// ---- 20_Product/10_BCF/11_Conv/12_E_Functions/01_DUTs/ST_CFG_Zone.TcDUT
// Zone configuration structure
TYPE ST_CFG_Zone:
(**************************************************************************************
 * 	Application		:	BoxControl Framework
 *	Revision		:	$Revision: 474969 $
 *	Revision date	:	$Date: 2021-04-08 19:53:18 +0200 (tor, 08 apr 2021) $
 *	Last changed by	:	$Author: d7mangc $
 *	URL				:	$URL: http://almscdc.swisslog.com/repo/SWPD/Development/BoxControlFramework/20_Release/tags/R1.12.0/01_Software/BCF/BCF/JumpStart/20_Product/10_BCF/11_Conv/12_E_Functions/01_DUTs/ST_CFG_Zone.TcDUT $
 *
 *	Purpose			:	Zone configuration - contains the configuration for a zone.
 *
 * ------------------------------------------------------------------------------------
 *	Copyright Swisslog [IP AG], Switzerland. All rights reserved.
 * 
 * ------------------------------------------------------------------------------------
 *	
 * 	Revision History: 
 *
 * VERSION DATE         INITIALS     DESCRIPTION
 * 0.0     DD.MM.YYYY   (name)       (explain customized modifications)
 *
 **************************************************************************************)
STRUCT
	ZoneName						: STRING[NAME_LENGTH]	:= 'MM-GGG-EEEE-FF-Z';			// Name of the zone
	Length							: ARRAY[1..3] OF UINT	:= [1000, 0, 0];				// Length of the zone based on the transport direction [mm]
	//-----------------------------------------------------------------------------------------------
	Speed							: REAL					:= 1.0;							// Maximal speed of the zone [m/s]
	SpeedSlow						: INT					:=  50;							// Speed slow [%]
	SpeedFast						: INT					:= 100;							// Speed fast [%]
	SpeedRatio						: REAL					:= 1/1;							// Transmission ratio between speed command and movement speed of the TU
	//-----------------------------------------------------------------------------------------------
	EnablePrestart					: BOOL					:= TRUE;						// Enable prestart drive two zones ahead
	EnableFreeRun					: BOOL					:= TRUE;						// Enable free run
	EnableMultipleTU_Transition		: BOOL					:= FALSE;						// Enable multiple TU transition
	EnableJamAutoReset				: BOOL					:= TRUE;						// Enable jam auto reset if signal is free
	EnableMFC						: BOOL					:= FALSE;						// Enable material flow control
	EnableIgnoreNextZoneState		: BOOL					:= FALSE;						// Enable ignore the state of the next zone at handover
	EnableSimultaneousTransport		: BOOL					:= FALSE;						// Enable simultaneous transport
	EnableLowPressureAccumulation	: BOOL					:= FALSE;						// Enable low pressure accumulation - NOT IMPLEMENTED -
	EnableSlugRelease				: BOOL					:= FALSE;						// Enable slug release -NOT IMPLEMENTED -
	EnableFastSpeed					: BOOL					:= TRUE;						// Enable fast speed 
	EnableMultizone					: BOOL					:= TRUE;						// Enable multizone
	EnableCreateGapOnlyAtRestart	: BOOL					:= FALSE;						// Enable create gap only when drive restarts
	EnableLatchOccupiedState		: BOOL					:= FALSE;						// Enable latch occupied state
	EnableRoutingUpdate             : BOOL                  := FALSE;						// Enable routing update
	EnableAddOnSensor               : BOOL    				:= FALSE;						// Will use the sensor from the addon interface
    EnableMotorControl              : BOOL                  := FALSE;                       // Needs to be enabled for the zones using common motor with slugging
	//-----------------------------------------------------------------------------------------------
	SendTransportTaskCompleted		: BOOL					:= FALSE;						// Send a transport complete report if destination is reached
	SendTransportTaskCompletedOcc	: BOOL					:= FALSE;						// Send a transport complete report if destination is reached and zone occupied
	SendPositionClear				: BOOL					:= FALSE;						// Send a position clear report if zone is physically free
	SendPositionOccupied			: BOOL					:= FALSE;						// Send a position pccupied report if zone is physically occupied
	SendIdentificationReport		: BOOL					:= FALSE;						// Send an identification point report if zone is physically occupied
	eTUR_SendMode					: E_TUR_SendModes		:= E_TUR_SendModes.ALWAYS;		// Additional controls over when TUR is sent on TU index deletion for the zone 
	//-----------------------------------------------------------------------------------------------
	AddTU_Data						: BOOL					:= FALSE;						// Add TU data 
	DeleteTU_DataTakeOver			: BOOL					:= FALSE;						// Delete TU data at takeover
	DeleteTU_DataZoneFree			: BOOL					:= FALSE;						// Delete TU data if the zone is free
	//-----------------------------------------------------------------------------------------------
	tZoneFree						: TIME					:= T#0S;						// Delay time for zone free, if 0 then standard value will be used (2s)
	tZoneOccupied					: TIME					:= T#0S;						// Delay time for zone occupied, if 0 then standard value will be used (2s)
	ClearingDistance				: UINT					:= 2_000;						// Clearing distance [mm]
	JamTriggerDistance				: UINT					:= 2_000;						// Driving distance after jam error is triggered [mm]
	TimeoutTakeDistance				: UINT					:= 0;							// Driving distance after timeout take is triggered, if 0 then calculated value will be used [mm]
	MinimumTU_Distance				: UINT					:= 0;							// Delays the takeover to ensure this minimum gap between the TU’s [mm]
	TakeoverPlausibilityDistance	: UINT					:= 0;							// Distance for takeover plausibility check, if 0 then calculated value will be used [mm] 
	StopDelayDistanceFromSide		: ARRAY[1..4] OF UINT	:= [  0,   0,   0,   0];		// Stop distance after occupied signal [mm]
    tTakeoverMotorStartDelay        : TIME                  := T#0S;						// Delay before starting the motor on takeover (slugging)
	ZoneEndLengthToSide				: ARRAY[1..4] OF UINT	:= [100, 100, 100, 100];		// Length between occupied signal and zone end [mm]
END_STRUCT
END_TYPE

// ---- 20_Product/10_BCF/11_Conv/12_E_Functions/01_DUTs/ST_CM_ZoneBase.TcDUT
TYPE ST_CM_ZoneBase :
(**************************************************************************************
 * 	Application		:	BoxControl Framework
 *	Revision		:	$Revision: 404529 $
 *	Revision date	:	$Date: 2018-04-23 08:21:38 +0200 (Mo., 23 Apr 2018) $
 *	Last changed by	:	$Author: b7bolm $
 *	URL				:	$URL: http://almscdc.swisslog.com/repo/SWPD/Development/BoxControlFramework/20_Release/trunk/01_Software/BCF/BCF/JumpStart/20_Product/10_App/12_E_Functions/10_Lib/10_Conv/01_DUTs/ST_CM_ZoneBase.TcDUT $
 *
 *	Purpose			:	Base Structure for Condition monitoring 					
 *
 *
 * ------------------------------------------------------------------------------------
 *	Copyright Swisslog [IP AG], Switzerland. All rights reserved.
 * 
 * ------------------------------------------------------------------------------------
 *	
 * 	Revision History: 
 *
 * 	VERSION			DATE			INITIALS			DESCRIPTION
 *	0.1				01.01.2001		swl					Example
 *
 **************************************************************************************)	
STRUCT
	nCurrentTime 	: ULINT; // Current DC-Time of the PLC-Task
	Data			: ARRAY[E_CM_Index.E_BEGIN_VARIABLE+1..E_CM_Index.E_END_VARIABLE-1] OF ST_CM_GeneralData; //Process Data used by Condiition Monitoring Method 
	Settings		: ARRAY[E_CM_Index.E_BEGIN_VARIABLE+1..E_CM_Index.E_END_VARIABLE-1] OF ST_CM_Settings; //Settings Data set by Telegram/User
	
END_STRUCT
END_TYPE

// ---- 20_Product/10_BCF/11_Conv/12_E_Functions/01_DUTs/ST_FunctionBase.TcDUT
TYPE ST_FunctionBase :
(**************************************************************************************
 * 	Application		:	BoxControl Framework
 *	Revision		:	$Revision: 404529 $
 *	Revision date	:	$Date: 2018-04-23 08:21:38 +0200 (Mo., 23 Apr 2018) $
 *	Last changed by	:	$Author: b7bolm $
 *	URL				:	$URL: http://almscdc.swisslog.com/repo/SWPD/Development/BoxControlFramework/20_Release/trunk/01_Software/BCF/BCF/JumpStart/20_Product/10_App/12_E_Functions/10_Lib/10_Conv/01_DUTs/ST_FunctionBase.TcDUT $
 *
 *	Purpose			:	Function interface - Contains data which is provided by the
 *						function or is input from other objects.
 *
 * ------------------------------------------------------------------------------------
 *	Copyright Swisslog [IP AG], Switzerland. All rights reserved.
 * 
 * ------------------------------------------------------------------------------------
 *	
 * 	Revision History: 
 *
 * 	VERSION			DATE			INITIALS			DESCRIPTION
 *	0.1				01.01.2001		swl					Example
 *
 **************************************************************************************)
STRUCT
	AddOnAck					: BOOL; // Addon acknowledge
	STI_Instance				: ITF_SubsystemTransport; // Instance to compare valid interfaces
	eMsgType					: E_ITC_MsgTypeConv;
	Position					: ST_PositionIdent; // Position idents
	NextPositionName			: STRING(NAME_LENGTH); // Position idents
	PrevPositionName			: STRING(NAME_LENGTH); // Position idents
	PositionName				: STRING(NAME_LENGTH); // Position name
	DestinationName				: STRING(NAME_LENGTH); // Position name
	TU_DataIndex				: DINT; // Data index
	ErrorDataSet				: ST_ErrorDataSet; // Temporary error set
	ErrorDataZone				: ST_ZoneErrorStruct; // Temporary error data
	eReturnCode					: E_ErrorConv;
	DataITC						: ST_ITC_GeneralData; // ITC Message
	OperatingState				: ST_PositionState; // States
	LinkedFunctionStopped		: BOOL; // Linked function stopped
	AllZonesStopped				: BOOL; // All zones are stopped
	TransportControlParam		: ST_TransportControlParam; // Transportcontrol param
	TransportData				: ST_TransportData; // Transport data
	PrevTransportData			: ST_TransportData; // Previous data
	NextTransportData			: ST_TransportData; // Next data
	TransportDataEmpty			: ST_TransportData; // Transport data
	TransportControlDataEmpty 	: ST_TransportControlData; // Transport control data
	ZoneSettingsEmpty			: ST_CFG_Zone; // Zone settings
	PositionStateEmpty			: ST_PositionState;
	Idx							: INT; // iterator
	FSQ							: ST_ITC_FSQ; // ITC Message
	FCQ							: ST_ITC_FCQ; // ITC Message
	MCQ							: ST_ITC_MCQ; // ITC Message
	SIQ							: ST_ITC_SIQ; // ITC Message
	DAQ							: ST_ITC_DAQ; // ITC Message
	GDQ							: ST_ITC_GDQ; // ITC Message
	RAA							: ST_ITC_RAA; // ITC Message
	RDQ							: ST_ITC_RDQ; // ITC Message
	CM_Zone						: ARRAY [1..NUMBER_OF_ZONES_PER_FUNCTION] OF ST_CM_Base;	/// Data Aquisition Variables Staorage and Settings // CM inside base
END_STRUCT
END_TYPE

// ---- 20_Product/10_BCF/11_Conv/12_E_Functions/01_DUTs/ST_FunctionData.TcDUT
TYPE ST_FunctionData :
(**************************************************************************************
 * 	Application		:	BoxControl Framework
 *	Revision		:	$Revision: 404529 $
 *	Revision date	:	$Date: 2018-04-23 08:21:38 +0200 (Mo., 23 Apr 2018) $
 *	Last changed by	:	$Author: b7bolm $
 *	URL				:	$URL: http://almscdc.swisslog.com/repo/SWPD/Development/BoxControlFramework/20_Release/trunk/01_Software/BCF/BCF/JumpStart/20_Product/10_App/12_E_Functions/10_Lib/10_Conv/01_DUTs/ST_FunctionData.TcDUT $
 *
 *	Purpose			:	Function data
 *
 * ------------------------------------------------------------------------------------
 *	Copyright Swisslog [IP AG], Switzerland. All rights reserved.
 * 
 * ------------------------------------------------------------------------------------
 *	
 * 	Revision History: 
 *
 * 	VERSION			DATE			INITIALS			DESCRIPTION
 *	0.1				01.01.2001		swl					Example
 *
 **************************************************************************************)
STRUCT
	Init				: BOOL; // Initialized
	InitRunning			: BOOL; // Init ongoing
	OperationState		: ST_PositionState; // Information about the state
	AddOn				: ST_AddOnResult; // Result form external addons
	MemberList			: ST_FunctionMemberList; // List of members belonging to this function
	ErrorData			: ST_FunctionErrorStruct; // Error structure
	AddOnData			: ST_AddOnData; // Specific addon data structs
	ControlRequest		: ST_ControlRequest; // Control request
END_STRUCT
END_TYPE

// ---- 20_Product/10_BCF/11_Conv/12_E_Functions/01_DUTs/ST_FunctionElement.TcDUT
TYPE ST_FunctionElement :
(**************************************************************************************
 * 	Application		:	BoxControl Framework
 *	Revision		:	$Revision: 404529 $
 *	Revision date	:	$Date: 2018-04-23 08:21:38 +0200 (Mo., 23 Apr 2018) $
 *	Last changed by	:	$Author: b7bolm $
 *	URL				:	$URL: http://almscdc.swisslog.com/repo/SWPD/Development/BoxControlFramework/20_Release/trunk/01_Software/BCF/BCF/JumpStart/20_Product/10_App/12_E_Functions/10_Lib/10_Conv/01_DUTs/ST_FunctionElement.TcDUT $
 *
 *	Purpose			:	Function element
 *
 * ------------------------------------------------------------------------------------
 *	Copyright Swisslog [IP AG], Switzerland. All rights reserved.
 * 
 * ------------------------------------------------------------------------------------
 *	
 * 	Revision History: 
 *
 * 	VERSION			DATE			INITIALS			DESCRIPTION
 *	0.1				01.01.2001		swl					Example
 *
 **************************************************************************************)	
STRUCT
	OperationState	: ST_PositionState;
	State			: ST_ElementState;
END_STRUCT
END_TYPE

// ---- 20_Product/10_BCF/11_Conv/12_E_Functions/01_DUTs/ST_FunctionErrorStruct.TcDUT
TYPE ST_FunctionErrorStruct :
(**************************************************************************************
 * 	Application		:	BoxControl Framework
 *	Revision		:	$Revision: 404529 $
 *	Revision date	:	$Date: 2018-04-23 08:21:38 +0200 (Mo., 23 Apr 2018) $
 *	Last changed by	:	$Author: b7bolm $
 *	URL				:	$URL: http://almscdc.swisslog.com/repo/SWPD/Development/BoxControlFramework/20_Release/trunk/01_Software/BCF/BCF/JumpStart/20_Product/10_App/12_E_Functions/10_Lib/10_Conv/01_DUTs/ST_FunctionErrorStruct.TcDUT $
 *
 *	Purpose			:	Function error structure - Contains all information for the
 *						error handling.
 *
 * ------------------------------------------------------------------------------------
 *	Copyright Swisslog [IP AG], Switzerland. All rights reserved.
 * 
 * ------------------------------------------------------------------------------------
 *	
 * 	Revision History: 
 *
 * 	VERSION			DATE			INITIALS			DESCRIPTION
 *	0.1				01.01.2001		swl					Example
 *
 **************************************************************************************)
STRUCT
	ErrorState				: E_ErrorState; // Ongoing module error state
	Error					: ST_ErrorDataSet; // Ongoing reported function error
	DataSetIdx				: INT; // Choosen error set index
	ErrorDataSet			: ARRAY [1..NUMBER_OF_ERROR_SETS] OF ST_ErrorDataSet; // Overview about all message sets
	ExternalError			: ST_ErrorDataSet; // External error, Can be set customized or by control code
	ZoneErrorPending		: BOOL; // A zone of this function is in error state
END_STRUCT
END_TYPE

// ---- 20_Product/10_BCF/11_Conv/12_E_Functions/01_DUTs/ST_FunctionInterface.TcDUT
TYPE ST_FunctionInterface :
(**************************************************************************************
 * 	Application		:	BoxControl Framework
 *	Revision		:	$Revision: 404529 $
 *	Revision date	:	$Date: 2018-04-23 08:21:38 +0200 (Mo., 23 Apr 2018) $
 *	Last changed by	:	$Author: b7bolm $
 *	URL				:	$URL: http://almscdc.swisslog.com/repo/SWPD/Development/BoxControlFramework/20_Release/trunk/01_Software/BCF/BCF/JumpStart/20_Product/10_App/12_E_Functions/10_Lib/10_Conv/01_DUTs/ST_FunctionInterface.TcDUT $
 *
 *	Purpose			:	Function interface - Contains data which is provided by the
 *						function or is input from other objects.
 *
 * ------------------------------------------------------------------------------------
 *	Copyright Swisslog [IP AG], Switzerland. All rights reserved.
 * 
 * ------------------------------------------------------------------------------------
 *	
 * 	Revision History: 
 *
 * 	VERSION			DATE			INITIALS			DESCRIPTION
 *	0.1				01.01.2001		swl					Example
 *
 **************************************************************************************)
STRUCT
	In		: ST_FunctionInterfaceIn;
	Out		: ST_FunctionInterfaceOut;
END_STRUCT
END_TYPE

// ---- 20_Product/10_BCF/11_Conv/12_E_Functions/01_DUTs/ST_FunctionInterfaceIn.TcDUT
TYPE ST_FunctionInterfaceIn :
(**************************************************************************************
 * 	Application		:	BoxControl Framework
 *	Revision		:	$Revision: 404529 $
 *	Revision date	:	$Date: 2018-04-23 08:21:38 +0200 (Mo., 23 Apr 2018) $
 *	Last changed by	:	$Author: b7bolm $
 *	URL				:	$URL: http://almscdc.swisslog.com/repo/SWPD/Development/BoxControlFramework/20_Release/trunk/01_Software/BCF/BCF/JumpStart/20_Product/10_App/12_E_Functions/10_Lib/10_Conv/01_DUTs/ST_FunctionInterfaceIn.TcDUT $
 *
 *	Purpose			:	Function interface - Contains data which is provided by the
 *						function or is input from other objects.
 *
 * ------------------------------------------------------------------------------------
 *	Copyright Swisslog [IP AG], Switzerland. All rights reserved.
 * 
 * ------------------------------------------------------------------------------------
 *	
 * 	Revision History: 
 *
 * 	VERSION			DATE			INITIALS			DESCRIPTION
 *	0.1				01.01.2001		swl					Example
 *
 **************************************************************************************)
STRUCT
	ePrevFunctionNumber 	: E_FunctionNumber; // Previous element function number
	eNextFunctionNumber 	: E_FunctionNumber; // Next element function number	
	FunctionEnable			: BOOL := TRUE; // External function enable 
	Element					: ST_FunctionElement; // States of the function corresponding element
	AddOnOrder				: ARRAY [1..Conveyor.NUMBER_OF_ADDON_FUNCTIONS] OF ST_AddOn; // Number of addons per function
END_STRUCT
END_TYPE

// ---- 20_Product/10_BCF/11_Conv/12_E_Functions/01_DUTs/ST_FunctionInterfaceOut.TcDUT
TYPE ST_FunctionInterfaceOut :
(**************************************************************************************
 * 	Application		:	BoxControl Framework
 *	Revision		:	$Revision: 404529 $
 *	Revision date	:	$Date: 2018-04-23 08:21:38 +0200 (Mo., 23 Apr 2018) $
 *	Last changed by	:	$Author: b7bolm $
 *	URL				:	$URL: http://almscdc.swisslog.com/repo/SWPD/Development/BoxControlFramework/20_Release/trunk/01_Software/BCF/BCF/JumpStart/20_Product/10_App/12_E_Functions/10_Lib/10_Conv/01_DUTs/ST_FunctionInterfaceOut.TcDUT $
 *
 *	Purpose			:	Function interface - Contains data which is provided by the
 *						function or is input from other objects.
 *
 * ------------------------------------------------------------------------------------
 *	Copyright Swisslog [IP AG], Switzerland. All rights reserved.
 * 
 * ------------------------------------------------------------------------------------
 *	
 * 	Revision History: 
 *
 * 	VERSION			DATE			INITIALS			DESCRIPTION
 *	0.1				01.01.2001		swl					Example
 *
 **************************************************************************************)
STRUCT
	FunctionOrders		: ST_FunctionOrders; // Function orders to the element
	AddOnOrders			: ST_AddOnOrders; // AddOn orders
	Interlock			: ST_Interlock; // Interlock structure
END_STRUCT
END_TYPE

// ---- 20_Product/10_BCF/11_Conv/12_E_Functions/01_DUTs/ST_FunctionMemberList.TcDUT
TYPE ST_FunctionMemberList :
(**************************************************************************************
 * 	Application		:	BoxControl Framework
 *	Revision		:	$Revision: 404529 $
 *	Revision date	:	$Date: 2018-04-23 08:21:38 +0200 (Mo., 23 Apr 2018) $
 *	Last changed by	:	$Author: b7bolm $
 *	URL				:	$URL: http://almscdc.swisslog.com/repo/SWPD/Development/BoxControlFramework/20_Release/trunk/01_Software/BCF/BCF/JumpStart/20_Product/10_App/12_E_Functions/10_Lib/10_Conv/01_DUTs/ST_FunctionMemberList.TcDUT $
 *
 *	Purpose			:	Function member list - Contains all objects belonging to this 
 *						function.
 *
 * ------------------------------------------------------------------------------------
 *	Copyright Swisslog [IP AG], Switzerland. All rights reserved.
 * 
 * ------------------------------------------------------------------------------------
 *	
 * 	Revision History: 
 *
 * 	VERSION			DATE			INITIALS			DESCRIPTION
 *	0.1				01.01.2001		swl					Example
 *
 **************************************************************************************)
STRUCT
	AddOnList		: ARRAY [1 .. NUMBER_OF_ADDON_FUNCTIONS] OF ST_AddonEntry;
END_STRUCT
END_TYPE

// ---- 20_Product/10_BCF/11_Conv/12_E_Functions/01_DUTs/ST_FunctionOrders.TcDUT
///Element function order - This structure serves as order command to the function related element.
TYPE ST_FunctionOrders :
(**************************************************************************************
 *  Application     :   BoxControl Framework
 *  Revision date   :   $Date: 2013-09-23 11:26:06 +0200 (Wed, 23 Sep 2015) $
 *  Author          :   CDC
 * ------------------------------------------------------------------------------------
 *  © Swisslog AG
 *  Swisslog is not liable for any usage of this source code that is not agreed 
 *  on between Swisslog and the other party. The mandatory legal liability remains 
 *  unaffected.
 * ------------------------------------------------------------------------------------
 *  Revision History: 
 *
 *  VERSION DATE         INITIALS     DESCRIPTION
 *  0.0     DD.MM.YYYY   (name)       (explain customized modifications)
 *
 **************************************************************************************)
 //Comment changed according to BCFD-6292 - ST_FunctionOrders, Comments not correct	
STRUCT
    //Axis 1 <-> 2
	Enable				: BOOL; // Function enables transport
	ReqDriveRun			: BOOL; // Request for drive run
	ReqDriveDirection	    : BOOL; // Request drive direction. TRUE = 1->2, False 2->1
	ReqSpeed			: INT; // Request for this speed

    //Axis 3 <-> 4
	Enable_34				: BOOL; // Function enables transport
	ReqDriveRun_34			: BOOL; // Request for drive run
	ReqSpeed_34				: INT; // Request for speed	
	ReqDriveDirection_34	: BOOL; // Request drive direction. True = 3->4, False = 4->3
END_STRUCT
END_TYPE

// ---- 20_Product/10_BCF/11_Conv/12_E_Functions/01_DUTs/ST_ITC_Function.TcDUT
TYPE ST_ITC_Function :
(**************************************************************************************
 * 	Application		:	BoxControl Framework
 *	Revision		:	$Revision: 404529 $
 *	Revision date	:	$Date: 2018-04-23 08:21:38 +0200 (Mo., 23 Apr 2018) $
 *	Last changed by	:	$Author: b7bolm $
 *	URL				:	$URL: http://almscdc.swisslog.com/repo/SWPD/Development/BoxControlFramework/20_Release/trunk/01_Software/BCF/BCF/JumpStart/20_Product/10_App/12_E_Functions/10_Lib/10_Conv/01_DUTs/ST_ITC_Function.TcDUT $
 *
 *	Purpose			:	Function ITC structure
 *
 * ------------------------------------------------------------------------------------
 *	Copyright Swisslog [IP AG], Switzerland. All rights reserved.
 * 
 * ------------------------------------------------------------------------------------
 *	
 * 	Revision History: 
 *
 * 	VERSION			DATE			INITIALS			DESCRIPTION
 *	0.1				01.01.2001		swl					Example
 *
 **************************************************************************************)
STRUCT
	FunctionITC		: ST_ITC_FunctionITC; // ITC function data
	ZoneITC			: ARRAY [1..NUMBER_OF_ZONES_PER_FUNCTION] OF ST_ITC_Zone; // ITC Zone data
	ManualMotion	: ST_ITC_ManualMotion; // Command for manual motion
END_STRUCT
END_TYPE

// ---- 20_Product/10_BCF/11_Conv/12_E_Functions/01_DUTs/ST_ITC_FunctionCommands.TcDUT
TYPE ST_ITC_FunctionCommands :
(**************************************************************************************
 * 	Application		:	BoxControl Framework
 *	Revision		:	$Revision: 404529 $
 *	Revision date	:	$Date: 2018-04-23 08:21:38 +0200 (Mo., 23 Apr 2018) $
 *	Last changed by	:	$Author: b7bolm $
 *	URL				:	$URL: http://almscdc.swisslog.com/repo/SWPD/Development/BoxControlFramework/20_Release/trunk/01_Software/BCF/BCF/JumpStart/20_Product/10_App/12_E_Functions/10_Lib/10_Conv/01_DUTs/ST_ITC_FunctionCommands.TcDUT $
 *
 *	Purpose			:	Internal ITC function commands
 *
 * ------------------------------------------------------------------------------------
 *	Copyright Swisslog [IP AG], Switzerland. All rights reserved.
 * 
 * ------------------------------------------------------------------------------------
 *	
 * 	Revision History: 
 *
 * 	VERSION			DATE			INITIALS			DESCRIPTION
 *	0.1				01.01.2001		swl					Example
 *
 **************************************************************************************)
STRUCT
	StatusReport			: BOOL; // Command to send StatusReport 
	ControlReport			: BOOL; // Command to send ControlReport 
	NoErrorReport			: BOOL; // Command to send a 'no error' report
	ManualControlReport		: BOOL; // Command to send a manual control report
	ScannerInformationReport: BOOL; // Command to send a scanner information report
	ScannerNoReadReport		: BOOL; // Command to send a scanner no read report
END_STRUCT
END_TYPE

// ---- 20_Product/10_BCF/11_Conv/12_E_Functions/01_DUTs/ST_ITC_FunctionITC.TcDUT
TYPE ST_ITC_FunctionITC :
(**************************************************************************************
 * 	Application		:	BoxControl Framework
 *	Revision		:	$Revision: 404529 $
 *	Revision date	:	$Date: 2018-04-23 08:21:38 +0200 (Mo., 23 Apr 2018) $
 *	Last changed by	:	$Author: b7bolm $
 *	URL				:	$URL: http://almscdc.swisslog.com/repo/SWPD/Development/BoxControlFramework/20_Release/trunk/01_Software/BCF/BCF/JumpStart/20_Product/10_App/12_E_Functions/10_Lib/10_Conv/01_DUTs/ST_ITC_FunctionITC.TcDUT $
 *
 *	Purpose			:	Function ITC structure
 *
 * ------------------------------------------------------------------------------------
 *	Copyright Swisslog [IP AG], Switzerland. All rights reserved.
 * 
 * ------------------------------------------------------------------------------------
 *	
 * 	Revision History: 
 *
 * 	VERSION			DATE			INITIALS			DESCRIPTION
 *	0.1				01.01.2001		swl					Example
 *
 **************************************************************************************)
STRUCT
	Commands		: ST_ITC_FunctionCommands; // Internal ITC commands
	Variable		: DINT; // Control variable
END_STRUCT
END_TYPE

// ---- 20_Product/10_BCF/11_Conv/12_E_Functions/01_DUTs/ST_ITC_Zone.TcDUT
TYPE ST_ITC_Zone :
(**************************************************************************************
 * 	Application		:	BoxControl Framework
 *	Revision		:	$Revision: 404529 $
 *	Revision date	:	$Date: 2018-04-23 08:21:38 +0200 (Mo., 23 Apr 2018) $
 *	Last changed by	:	$Author: b7bolm $
 *	URL				:	$URL: http://almscdc.swisslog.com/repo/SWPD/Development/BoxControlFramework/20_Release/trunk/01_Software/BCF/BCF/JumpStart/20_Product/10_App/12_E_Functions/10_Lib/10_Conv/01_DUTs/ST_ITC_Zone.TcDUT $
 *
 *	Purpose			:	Zone ITC structures
 *
 * ------------------------------------------------------------------------------------
 *	Copyright Swisslog [IP AG], Switzerland. All rights reserved.
 * 
 * ------------------------------------------------------------------------------------
 *	
 * 	Revision History: 
 *
 * 	VERSION			DATE			INITIALS			DESCRIPTION
 *	0.1				01.01.2001		swl					Example
 *
 **************************************************************************************)
STRUCT
	Commands	: ST_ITC_ZoneCommands; // Internal zone ITC commands
	Variable	: DINT; // Control variable
	Flags		: ST_ITC_ZoneFlags; // Flags
END_STRUCT
END_TYPE

// ---- 20_Product/10_BCF/11_Conv/12_E_Functions/01_DUTs/ST_ITC_ZoneCommands.TcDUT
TYPE ST_ITC_ZoneCommands :
(**************************************************************************************
 * 	Application		:	BoxControl Framework
 *	Revision		:	$Revision: 404529 $
 *	Revision date	:	$Date: 2018-04-23 08:21:38 +0200 (Mo., 23 Apr 2018) $
 *	Last changed by	:	$Author: b7bolm $
 *	URL				:	$URL: http://almscdc.swisslog.com/repo/SWPD/Development/BoxControlFramework/20_Release/trunk/01_Software/BCF/BCF/JumpStart/20_Product/10_App/12_E_Functions/10_Lib/10_Conv/01_DUTs/ST_ITC_ZoneCommands.TcDUT $
 *
 *	Purpose			:	Zone commands
 *
 * ------------------------------------------------------------------------------------
 *	Copyright Swisslog [IP AG], Switzerland. All rights reserved.
 * 
 * ------------------------------------------------------------------------------------
 *	
 * 	Revision History: 
 *
 * 	VERSION			DATE			INITIALS			DESCRIPTION
 *	0.1				01.01.2001		swl					Example
 *
 **************************************************************************************)	
STRUCT
	NoErrorReport				: BOOL; // Command to send a no error report 
	StatusReport				: BOOL; // Command to send a status report 
	ControlReport				: BOOL; // Command TO send a control report 
	TransportTaskCompleted		: BOOL; // Command to send a transport task report 
	PositionOccupied			: BOOL; // Command to send a position occupied report 
	PositionCleared				: BOOL; // Command to send a position cleared report 
	IdentificationReport		: BOOL; // Command to send an identification point report
END_STRUCT
END_TYPE

// ---- 20_Product/10_BCF/11_Conv/12_E_Functions/01_DUTs/ST_ITC_ZoneFlags.TcDUT
TYPE ST_ITC_ZoneFlags :
(**************************************************************************************
 * 	Application		:	BoxControl Framework
 *	Revision		:	$Revision: 404529 $
 *	Revision date	:	$Date: 2018-04-23 08:21:38 +0200 (Mo., 23 Apr 2018) $
 *	Last changed by	:	$Author: b7bolm $
 *	URL				:	$URL: http://almscdc.swisslog.com/repo/SWPD/Development/BoxControlFramework/20_Release/trunk/01_Software/BCF/BCF/JumpStart/20_Product/10_App/12_E_Functions/10_Lib/10_Conv/01_DUTs/ST_ITC_ZoneFlags.TcDUT $
 *
 *	Purpose			:	Zone flags
 *
 * ------------------------------------------------------------------------------------
 *	Copyright Swisslog [IP AG], Switzerland. All rights reserved.
 * 
 * ------------------------------------------------------------------------------------
 *	
 * 	Revision History: 
 *
 * 	VERSION			DATE			INITIALS			DESCRIPTION
 *	0.1				01.01.2001		swl					Example
 *
 **************************************************************************************)	
STRUCT
	TransportTaksCompleteOccSent	: BOOL; // Store sent information
	TransportTaksCompleteSent		: BOOL; // Store sent information
	PositionClearSent				: BOOL; // Store sent information
	PositionOccupiedSent			: BOOL; // Store sent information
	IdentificationReportSent		: BOOL; // Store sent information
END_STRUCT
END_TYPE

// ---- 20_Product/10_BCF/11_Conv/12_E_Functions/01_DUTs/ST_LastTUdata.TcDUT
TYPE ST_LastTUdata :
STRUCT
	TU_ID			: STRING(Conveyor.TU_ID_STRINGLENGTH); // TU_ID as characters 1 to 18 
  	AssignmentID	: UDINT; // Assignment ID
  	TU_Type			: INT; // Type of transport unit 
END_STRUCT
END_TYPE

// ---- 20_Product/10_BCF/11_Conv/12_E_Functions/01_DUTs/ST_TransportControlData.TcDUT
TYPE ST_TransportControlData :
(**************************************************************************************
 * 	Application		:	BoxControl Framework
 *	Revision		:	$Revision: 404529 $
 *	Revision date	:	$Date: 2018-04-23 08:21:38 +0200 (Mo., 23 Apr 2018) $
 *	Last changed by	:	$Author: b7bolm $
 *	URL				:	$URL: http://almscdc.swisslog.com/repo/SWPD/Development/BoxControlFramework/20_Release/trunk/01_Software/BCF/BCF/JumpStart/20_Product/10_App/12_E_Functions/10_Lib/10_Conv/01_DUTs/ST_TransportControlData.TcDUT $
 *
 *	Purpose			:	Transport control
 *
 * ------------------------------------------------------------------------------------
 *	Copyright Swisslog [IP AG], Switzerland. All rights reserved.
 * 
 * ------------------------------------------------------------------------------------
 *	
 * 	Revision History: 
 *
 * 	VERSION			DATE			INITIALS			DESCRIPTION
 *	0.1				01.01.2001		swl					Example
 *
 **************************************************************************************)	
STRUCT
	eTransportState					: E_TransportState		:= E_TransportState.UNDEFINED;	// Transport state
	eTakeOverState 					: E_TakeOverState		:= E_TakeOverState.UNDEFINED;	// Takeover state
	eHandOverState 					: E_HandOverState		:= E_HandOverState.UNDEFINED;	// Handover state
	TransportParam					: ST_TransportParam;									// Transport parameter valid for current transport
	//-----------------------------------------------------------------------------------------------
	Occupied						: BOOL					:= FALSE; 						// Position is physically occupied
	DataPresent						: BOOL					:= FALSE;						// Position is logically occupied
	TU_DataIndex					: DINT					:= 0;							// Current TU data index
	LastTU_DataIndex 				: DINT					:= 0;							// Last TU data index
	NumberOfPresentTUs  			: UINT					:= 0;							// Number of present TUs on this zone (the TU in handover is counted by the next zone)
	FastSpeedActive					: BOOL					:= FALSE;						// Fast speed is active
	DriveRunning					: BOOL					:= FALSE;						// Drive is running
	MovementPosition				: UDINT					:= 0;							// Movement position value [mm]	
	Stopped							: BOOL					:= FALSE;						// Module is stopped
	SensorOccupied      			: BOOL					:= FALSE;						// Sensor position occupied
	TransportActive     			: BOOL					:= FALSE;						// Transport is active
	//-----------------------------------------------------------------------------------------------
	CurrentSpeed					: INT					:= 0;							// Current speed
	LimitSpeedToPrev				: INT					:= 0;							// Current valid speed limit to previous zone
	LimitSpeedToNext				: INT					:= 0;							// Current valid speed limit to next zone
	//-----------------------------------------------------------------------------------------------
	TU_LeadingEdgePos				: DINT					:= 0;							// TU leading edge position [mm]
END_STRUCT
END_TYPE

// ---- 20_Product/10_BCF/11_Conv/12_E_Functions/01_DUTs/ST_TransportControlParam.TcDUT
TYPE ST_TransportControlParam :
(**************************************************************************************
 * 	Application		:	BoxControl Framework
 *	Revision		:	$Revision: 404529 $
 *	Revision date	:	$Date: 2018-04-23 08:21:38 +0200 (Mo., 23 Apr 2018) $
 *	Last changed by	:	$Author: b7bolm $
 *	URL				:	$URL: http://almscdc.swisslog.com/repo/SWPD/Development/BoxControlFramework/20_Release/trunk/01_Software/BCF/BCF/JumpStart/20_Product/10_App/12_E_Functions/10_Lib/10_Conv/01_DUTs/ST_TransportControlParam.TcDUT $
 *
 *	Purpose			:	Transport control parameter
 *
 * ------------------------------------------------------------------------------------
 *	Copyright Swisslog [IP AG], Switzerland. All rights reserved.
 * 
 * ------------------------------------------------------------------------------------
 *	
 * 	Revision History: 
 *
 * 	VERSION			DATE			INITIALS			DESCRIPTION
 *	0.1				01.01.2001		swl					Example
 *
 **************************************************************************************)	
STRUCT
	reFunctionNumber			: REFERENCE TO E_FunctionNumber; // Number oft the function
	rOperationState				: REFERENCE TO ST_PositionState; // Function state
	rePrevFunctionNumber		: REFERENCE TO E_FunctionNumber; // Previous function number
	reNextFunctionNumber		: REFERENCE TO E_FunctionNumber; // Next function number
	ZoneNumber 				    : INT; // Number of the zone
	rSettings 					: REFERENCE TO ST_CFG_Zone; // Settings of the zone
	reSetFuncPrevFuncNumber  	: REFERENCE TO E_FunctionNumber; // Settings function previous function number
	reSetFuncNextFuncNumber  	: REFERENCE TO E_FunctionNumber; // Settings function next function number
	rZoneEnable      			: REFERENCE TO ST_TransportEnable; // Zone enable
	rExternalZoneEnable 		: REFERENCE TO BOOL; // External enable 
END_STRUCT
END_TYPE

// ---- 20_Product/10_BCF/11_Conv/12_E_Functions/01_DUTs/ST_TransportControl_Inputs.TcDUT
TYPE ST_TransportControl_Inputs :
(**************************************************************************************
 * 	Application		:	BoxControl Framework
 *	Revision		:	$Revision: 404529 $
 *	Revision date	:	$Date: 2018-04-23 08:21:38 +0200 (Mo., 23 Apr 2018) $
 *	Last changed by	:	$Author: b7bolm $
 *	URL				:	$URL: http://almscdc.swisslog.com/repo/SWPD/Development/BoxControlFramework/20_Release/trunk/01_Software/BCF/BCF/JumpStart/20_Product/10_App/12_E_Functions/10_Lib/10_Conv/10_Functions/01_DUTs/ST_TransportControl_Inputs.TcDUT $
 *
 *	Purpose			:	Transport control inputs
 *
 * ------------------------------------------------------------------------------------
 *	Copyright Swisslog [IP AG], Switzerland. All rights reserved.
 * 
 * ------------------------------------------------------------------------------------
 *	
 * 	Revision History: 
 *
 * 	VERSION			DATE			INITIALS			DESCRIPTION
 *	0.1				01.01.2001		swl					Example
 *
 **************************************************************************************)	
STRUCT
	Enable 		: ST_TransportEnable; // Transport enable
	MasterSpeed : INT; // Master speed of the Subsystem [%]
END_STRUCT
END_TYPE

// ---- 20_Product/10_BCF/11_Conv/12_E_Functions/01_DUTs/ST_TransportControl_Outputs.TcDUT
TYPE ST_TransportControl_Outputs :
(**************************************************************************************
 * 	Application		:	BoxControl Framework
 *	Revision		:	$Revision: 404529 $
 *	Revision date	:	$Date: 2018-04-23 08:21:38 +0200 (Mo., 23 Apr 2018) $
 *	Last changed by	:	$Author: b7bolm $
 *	URL				:	$URL: http://almscdc.swisslog.com/repo/SWPD/Development/BoxControlFramework/20_Release/trunk/01_Software/BCF/BCF/JumpStart/20_Product/10_App/12_E_Functions/10_Lib/10_Conv/10_Functions/01_DUTs/ST_TransportControl_Outputs.TcDUT $
 *
 *	Purpose			:	Transport control outputs
 *
 * ------------------------------------------------------------------------------------
 *	Copyright Swisslog [IP AG], Switzerland. All rights reserved.
 * 
 * ------------------------------------------------------------------------------------
 *	
 * 	Revision History: 
 *
 * 	VERSION			DATE			INITIALS			DESCRIPTION
 *	0.1				01.01.2001		swl					Example 
 *
 **************************************************************************************)	
STRUCT
	DriveRun   				 : BOOL; // Run signal for drive
	DriveTakeoverRun		 : BOOL; // Run signal for drive takeover
	DriveHandoverRun		 : BOOL; // Run signal for drive handover
	RequestPrevTransportData : BOOL; // Request previous transport data
	RequestNextTransportData : BOOL; // Request next transport data
	DeletePrevTransportData	 : BOOL; // Delete previous transport data
	DeleteNextTransportData  : BOOL; // Delete next transport data
	DistanceToZoneEnd		 : UINT; // Distance TU leading edge to zone end [mm]	
END_STRUCT
END_TYPE

// ---- 20_Product/10_BCF/11_Conv/12_E_Functions/01_DUTs/ST_TransportData.TcDUT
TYPE ST_TransportData :
(**************************************************************************************
 * 	Application		:	BoxControl Framework
 *	Revision		:	$Revision: 404529 $
 *	Revision date	:	$Date: 2018-04-23 08:21:38 +0200 (Mo., 23 Apr 2018) $
 *	Last changed by	:	$Author: b7bolm $
 *	URL				:	$URL: http://almscdc.swisslog.com/repo/SWPD/Development/BoxControlFramework/20_Release/trunk/01_Software/BCF/BCF/JumpStart/20_Product/10_App/12_E_Functions/10_Lib/10_Conv/01_DUTs/ST_TransportData.TcDUT $
 *
 *	Purpose			:	Transport control data
 *
 * ------------------------------------------------------------------------------------
 *	Copyright Swisslog [IP AG], Switzerland. All rights reserved.
 * 
 * ------------------------------------------------------------------------------------
 *	
 * 	Revision History: 
 *
 * 	VERSION			DATE			INITIALS			DESCRIPTION
 *	0.1				01.01.2001		swl					Example
 *
 **************************************************************************************)	
STRUCT
	eFunctionNumber			: E_FunctionNumber; // Number oft the function			
	ZoneNumber 				: INT;
	rSettings 				: REFERENCE TO ST_CFG_Zone;
	rTransportControlData	: REFERENCE TO ST_TransportControlData;
END_STRUCT
END_TYPE

// ---- 20_Product/10_BCF/11_Conv/12_E_Functions/01_DUTs/ST_TransportDataRequest.TcDUT
TYPE ST_TransportDataRequest :
(**************************************************************************************
 * 	Application		:	BoxControl Framework
 *	Revision		:	$Revision: 404529 $
 *	Revision date	:	$Date: 2018-04-23 08:21:38 +0200 (Mo., 23 Apr 2018) $
 *	Last changed by	:	$Author: b7bolm $
 *	URL				:	$URL: http://almscdc.swisslog.com/repo/SWPD/Development/BoxControlFramework/20_Release/trunk/01_Software/BCF/BCF/JumpStart/20_Product/10_App/12_E_Functions/10_Lib/10_Conv/10_Functions/01_DUTs/ST_TransportDataRequest.TcDUT $
 *
 *	Purpose			:	Transport control inputs
 *
 * ------------------------------------------------------------------------------------
 *	Copyright Swisslog [IP AG], Switzerland. All rights reserved.
 * 
 * ------------------------------------------------------------------------------------
 *	
 * 	Revision History: 
 *
 * 	VERSION			DATE			INITIALS			DESCRIPTION
 *	0.1				01.01.2001		swl					Example
 *
 **************************************************************************************)	
STRUCT
	RequestPrevTransportData : BOOL; // Request previous transport data
	RequestNextTransportData : BOOL; // Request next transport data
	DeletePrevTransportData	 : BOOL; // Delete previous transport data
	DeleteNextTransportData  : BOOL; // Delete next transport data
END_STRUCT
END_TYPE

// ---- 20_Product/10_BCF/11_Conv/12_E_Functions/01_DUTs/ST_TransportEnable.TcDUT
TYPE ST_TransportEnable :
(**************************************************************************************
 * 	Application		:	BoxControl Framework
 *	Revision		:	$Revision: 404529 $
 *	Revision date	:	$Date: 2018-04-23 08:21:38 +0200 (Mo., 23 Apr 2018) $
 *	Last changed by	:	$Author: b7bolm $
 *	URL				:	$URL: http://almscdc.swisslog.com/repo/SWPD/Development/BoxControlFramework/20_Release/trunk/01_Software/BCF/BCF/JumpStart/20_Product/10_App/12_E_Functions/10_Lib/10_Conv/01_DUTs/ST_TransportEnable.TcDUT $
 *
 *	Purpose			:	Transport enable
 *
 * ------------------------------------------------------------------------------------
 *	Copyright Swisslog [IP AG], Switzerland. All rights reserved.
 * 
 * ------------------------------------------------------------------------------------
 *	
 * 	Revision History: 
 *
 * 	VERSION			DATE			INITIALS			DESCRIPTION
 *	0.1				01.01.2001		swl					Example
 *
 **************************************************************************************)	
STRUCT
	Transport 	: BOOL := TRUE; // Enable transport general
	TakeOver 	: BOOL := TRUE; // Enable start transport takeover
	HandOver 	: BOOL := TRUE; // Enable start transport handover
END_STRUCT
END_TYPE

// ---- 20_Product/10_BCF/11_Conv/12_E_Functions/01_DUTs/ST_TransportParam.TcDUT
TYPE ST_TransportParam :
(**************************************************************************************
 * 	Application		:	BoxControl Framework
 *	Revision		:	$Revision: 404529 $
 *	Revision date	:	$Date: 2018-04-23 08:21:38 +0200 (Mo., 23 Apr 2018) $
 *	Last changed by	:	$Author: b7bolm $
 *	URL				:	$URL: http://almscdc.swisslog.com/repo/SWPD/Development/BoxControlFramework/20_Release/trunk/01_Software/BCF/BCF/JumpStart/20_Product/10_App/12_E_Functions/10_Lib/10_Conv/01_DUTs/ST_TransportParam.TcDUT $
 *
 *	Purpose			:	Transport parameter
 *
 * ------------------------------------------------------------------------------------
 *	Copyright Swisslog [IP AG], Switzerland. All rights reserved.
 * 
 * ------------------------------------------------------------------------------------
 *	
 * 	Revision History: 
 *
 * 	VERSION			DATE			INITIALS			DESCRIPTION
 *	0.1				01.01.2001		swl					Example
 *
 **************************************************************************************)	
STRUCT
	ZoneLength						: UINT					:= 0;							// Length of the zone [mm]
	StopDelayDistance				: UINT					:= 0;							// Stop distance after occupied signal [mm]
    ZoneEndLength 					: UINT					:= 0;							// Length between occupied signal and zone end [mm]
END_STRUCT
END_TYPE

// ---- 20_Product/10_BCF/11_Conv/12_E_Functions/01_DUTs/ST_ZoneData.TcDUT
TYPE ST_ZoneData :
(**************************************************************************************
 * 	Application		:	BoxControl Framework
 *	Revision		:	$Revision: 404529 $
 *	Revision date	:	$Date: 2018-04-23 08:21:38 +0200 (Mo., 23 Apr 2018) $
 *	Last changed by	:	$Author: b7bolm $
 *	URL				:	$URL: http://almscdc.swisslog.com/repo/SWPD/Development/BoxControlFramework/20_Release/trunk/01_Software/BCF/BCF/JumpStart/20_Product/10_App/12_E_Functions/10_Lib/10_Conv/01_DUTs/ST_ZoneData.TcDUT $
 *
 *	Purpose			:	Zone data
 *
 * ------------------------------------------------------------------------------------
 *	Copyright Swisslog [IP AG], Switzerland. All rights reserved.
 * 
 * ------------------------------------------------------------------------------------
 *	
 * 	Revision History: 
 *
 * 	VERSION			DATE			INITIALS			DESCRIPTION
 *	0.1				01.01.2001		swl					Example
 *
 **************************************************************************************)
STRUCT
	Init 					: BOOL; // Initialized
	InitRunning				: BOOL; // Initialization running
	AddOn					: ST_AddOnResult; // Valid addon result
	TransportControlData	: ST_TransportControlData; // Transport control data
	ErrorData				: ST_ZoneErrorStruct; // Error structure
	LastTUdata				: ST_LastTUdata; // Data from last TU on position
END_STRUCT
END_TYPE

// ---- 20_Product/10_BCF/11_Conv/12_E_Functions/01_DUTs/ST_ZoneErrorStruct.TcDUT
TYPE ST_ZoneErrorStruct :
(**************************************************************************************
 * 	Application		:	BoxControl Framework
 *	Revision		:	$Revision: 404529 $
 *	Revision date	:	$Date: 2018-04-23 08:21:38 +0200 (Mo., 23 Apr 2018) $
 *	Last changed by	:	$Author: b7bolm $
 *	URL				:	$URL: http://almscdc.swisslog.com/repo/SWPD/Development/BoxControlFramework/20_Release/trunk/01_Software/BCF/BCF/JumpStart/20_Product/10_App/12_E_Functions/10_Lib/10_Conv/01_DUTs/ST_ZoneErrorStruct.TcDUT $
 *
 *	Purpose			:	Zone error structure - Contains all information for the
 *						error handling.
 *
 * ------------------------------------------------------------------------------------
 *	Copyright Swisslog [IP AG], Switzerland. All rights reserved.
 * 
 * ------------------------------------------------------------------------------------
 *	
 * 	Revision History: 
 *
 * 	VERSION			DATE			INITIALS			DESCRIPTION
 *	0.1				01.01.2001		swl					Example
 *
 **************************************************************************************)
STRUCT
	ErrorState				: E_ErrorState; // Ongoing module error state
	Error					: ST_ErrorDataSet; // Ongoing reported function error
	DataSetIdx				: INT; // Choosen error set index
	ErrorDataSet			: ARRAY [1..NUMBER_OF_ERROR_SETS] OF ST_ErrorDataSet; // Overview about all message sets
	ExternalError			: ST_ErrorDataSet; // External error, Can be set customized or by control code
END_STRUCT
END_TYPE

// ---- 20_Product/10_BCF/11_Conv/12_E_Functions/01_DUTs/ST_ZoneInterface.TcDUT
TYPE ST_ZoneInterface :
(**************************************************************************************
 * 	Application		:	BoxControl Framework
 *	Revision		:	$Revision: 404529 $
 *	Revision date	:	$Date: 2018-04-23 08:21:38 +0200 (Mo., 23 Apr 2018) $
 *	Last changed by	:	$Author: b7bolm $
 *	URL				:	$URL: http://almscdc.swisslog.com/repo/SWPD/Development/BoxControlFramework/20_Release/trunk/01_Software/BCF/BCF/JumpStart/20_Product/10_App/12_E_Functions/10_Lib/10_Conv/01_DUTs/ST_ZoneInterface.TcDUT $
 *
 *	Purpose			:	Zone interface
 *
 * ------------------------------------------------------------------------------------
 *	Copyright Swisslog [IP AG], Switzerland. All rights reserved.
 * 
 * ------------------------------------------------------------------------------------
 *	
 * 	Revision History: 
 *
 * 	VERSION			DATE			INITIALS			DESCRIPTION
 *	0.1				01.01.2001		swl					Example
 *
 **************************************************************************************)	
STRUCT
	In		: ST_ZoneInterfaceIn;
	Out		: ST_ZoneInterfaceOut;
END_STRUCT
END_TYPE

// ---- 20_Product/10_BCF/11_Conv/12_E_Functions/01_DUTs/ST_ZoneInterfaceIn.TcDUT
TYPE ST_ZoneInterfaceIn :
(**************************************************************************************
 * 	Application		:	BoxControl Framework
 *	Revision		:	$Revision: 404529 $
 *	Revision date	:	$Date: 2018-04-23 08:21:38 +0200 (Mo., 23 Apr 2018) $
 *	Last changed by	:	$Author: b7bolm $
 *	URL				:	$URL: http://almscdc.swisslog.com/repo/SWPD/Development/BoxControlFramework/20_Release/trunk/01_Software/BCF/BCF/JumpStart/20_Product/10_App/12_E_Functions/10_Lib/10_Conv/01_DUTs/ST_ZoneInterfaceIn.TcDUT $
 *
 *	Purpose			:	Zone interface
 *
 * ------------------------------------------------------------------------------------
 *	Copyright Swisslog [IP AG], Switzerland. All rights reserved.
 * 
 * ------------------------------------------------------------------------------------
 *	
 * 	Revision History: 
 *
 * 	VERSION			DATE			INITIALS			DESCRIPTION
 *	0.1				01.01.2001		swl					Example
 *
 **************************************************************************************)	
STRUCT
	ZoneEnable 	: BOOL := TRUE; // Enable zone for external use
	Enable 		: ST_TransportEnable; // Zone enable
END_STRUCT
END_TYPE

// ---- 20_Product/10_BCF/11_Conv/12_E_Functions/01_DUTs/ST_ZoneInterfaceOut.TcDUT
TYPE ST_ZoneInterfaceOut :
(**************************************************************************************
 * 	Application		:	BoxControl Framework
 *	Revision		:	$Revision: 404529 $
 *	Revision date	:	$Date: 2018-04-23 08:21:38 +0200 (Mo., 23 Apr 2018) $
 *	Last changed by	:	$Author: b7bolm $
 *	URL				:	$URL: http://almscdc.swisslog.com/repo/SWPD/Development/BoxControlFramework/20_Release/trunk/01_Software/BCF/BCF/JumpStart/20_Product/10_App/12_E_Functions/10_Lib/10_Conv/01_DUTs/ST_ZoneInterfaceOut.TcDUT $
 *
 *	Purpose			:	Zone interface
 *
 * ------------------------------------------------------------------------------------
 *	Copyright Swisslog [IP AG], Switzerland. All rights reserved.
 * 
 * ------------------------------------------------------------------------------------
 *	
 * 	Revision History: 
 *
 * 	VERSION			DATE			INITIALS			DESCRIPTION
 *	0.1				01.01.2001		swl					Example
 *
 **************************************************************************************)	
STRUCT
	;
END_STRUCT
END_TYPE

// ---- 20_Product/10_BCF/11_Conv/13_Elements/01_DUTs/E_ElementType.TcDUT
TYPE E_ElementType :
(**************************************************************************************
 * 	Application		:	BoxControl Framework
 *	Revision		:	$Revision: 404529 $
 *	Revision date	:	$Date: 2018-04-23 08:21:38 +0200 (Mo., 23 Apr 2018) $
 *	Last changed by	:	$Author: b7bolm $
 *	URL				:	$URL: http://almscdc.swisslog.com/repo/SWPD/Development/BoxControlFramework/20_Release/trunk/01_Software/BCF/BCF/JumpStart/20_Product/10_App/13_Elements/10_Lib/10_Conv/01_DUTs/E_ElementType.TcDUT $
 *
 *	Purpose			:	Element type
 *
 * ------------------------------------------------------------------------------------
 *	Copyright Swisslog [IP AG], Switzerland. All rights reserved.
 * 
 * ------------------------------------------------------------------------------------
 *	
 * 	Revision History: 
 *
 * 	VERSION			DATE			INITIALS			DESCRIPTION
 *	0.1				01.01.2001		swl					Example
 *
 **************************************************************************************)	
(
	NO_TYPE
);
END_TYPE

// ---- 20_Product/10_BCF/11_Conv/13_Elements/01_DUTs/E_ITC_ElementControlCode.TcDUT
TYPE E_ITC_ElementControlCode :
(**************************************************************************************
 * 	Application		:	BoxControl Framework
 *	Revision		:	$Revision: 404529 $
 *	Revision date	:	$Date: 2018-04-23 08:21:38 +0200 (Mo., 23 Apr 2018) $
 *	Last changed by	:	$Author: b7bolm $
 *	URL				:	$URL: http://almscdc.swisslog.com/repo/SWPD/Development/BoxControlFramework/20_Release/trunk/01_Software/BCF/BCF/JumpStart/20_Product/10_App/13_Elements/10_Lib/10_Conv/01_DUTs/E_ITC_ElementControlCode.TcDUT $
 *
 *	Purpose			:	Element control code
 *
 * ------------------------------------------------------------------------------------
 *	Copyright Swisslog [IP AG], Switzerland. All rights reserved.
 * 
 * ------------------------------------------------------------------------------------
 *	
 * 	Revision History: 
 *
 * 	VERSION			DATE			INITIALS			DESCRIPTION
 *	0.1				01.01.2001		swl					Example
 *
 **************************************************************************************)
(
	NO_CODE					:= 0, // No code
	RESET_ERROR 			:= 1, // Acknowledge Error
	INITIALIZE				:= 2, // Initialize
	ENABLE					:= 4, // E.g. start, stop
	SET_VARIABLE			:= 5, // Set Variable
	SET_ERROR				:= 20 // Set error
);
END_TYPE

// ---- 20_Product/10_BCF/11_Conv/13_Elements/01_DUTs/ST_CFG_Element.TcDUT
TYPE ST_CFG_Element :
(**************************************************************************************
 * 	Application		:	BoxControl Framework
 *	Revision		:	$Revision: 404529 $
 *	Revision date	:	$Date: 2018-04-23 08:21:38 +0200 (Mo., 23 Apr 2018) $
 *	Last changed by	:	$Author: b7bolm $
 *	URL				:	$URL: http://almscdc.swisslog.com/repo/SWPD/Development/BoxControlFramework/20_Release/trunk/01_Software/BCF/BCF/JumpStart/20_Product/10_App/13_Elements/10_Lib/10_Conv/01_DUTs/10_Dummy/ST_CFG_Element.TcDUT $
 *
 *	Purpose			:	Base element configuration.
 *
 * ------------------------------------------------------------------------------------
 *	Copyright Swisslog [IP AG], Switzerland. All rights reserved.
 * 
 * ------------------------------------------------------------------------------------
 *	
 * 	Revision History: 
 *
 * 	VERSION			DATE			INITIALS			DESCRIPTION
 *	0.1				01.01.2001		swl					Example
 *
 **************************************************************************************)
STRUCT
	ElementName 			: STRING(NAME_LENGTH); // Element name as string
	eElementNumber			: E_ElementNumber; // Element number
	eElementType			: E_ElementType; // Element type
	eSlaveElementNumber		: E_ElementNumber; // Element slave
	eSlaveElementNumber_12	: E_ElementNumber; // Element slave
	eSlaveElementNumber_34	: E_ElementNumber; // Element slave
	eMasterElementNumber	: E_ElementNumber; // Element slave
	eMasterElementNumber_12	: E_ElementNumber; // Element slave
	eMasterElementNumber_34	: E_ElementNumber; // Element slave
END_STRUCT
END_TYPE

// ---- 20_Product/10_BCF/11_Conv/13_Elements/01_DUTs/ST_ElementBase.TcDUT
TYPE ST_ElementBase :
(**************************************************************************************
 * 	Application		:	BoxControl Framework
 *	Revision		:	$Revision: 404529 $
 *	Revision date	:	$Date: 2018-04-23 08:21:38 +0200 (Mo., 23 Apr 2018) $
 *	Last changed by	:	$Author: b7bolm $
 *	URL				:	$URL: http://almscdc.swisslog.com/repo/SWPD/Development/BoxControlFramework/20_Release/trunk/01_Software/BCF/BCF/JumpStart/20_Product/10_App/13_Elements/10_Lib/10_Conv/01_DUTs/ST_ElementBase.TcDUT $
 *
 *	Purpose			:	Basis element data
 *
 * ------------------------------------------------------------------------------------
 *	Copyright Swisslog [IP AG], Switzerland. All rights reserved.
 * 
 * ------------------------------------------------------------------------------------
 *	
 * 	Revision History: 
 *
 * 	VERSION			DATE			INITIALS			DESCRIPTION
 *	0.1				01.01.2001		swl					Example
 *
 **************************************************************************************)
STRUCT
	eMsgType				: E_ITC_MsgTypeConv; // ITC message
	eReturnCode				: E_ErrorConv; // Error code
	FunctionStopped			: BOOL; // Function are stopped
	Idx						: INT; // Iterator
	MemberState				: ST_PositionState; // Member state
	FunctionOrdersEmpty		: ST_FunctionOrders;
	OperationStateEmpty		: ST_PositionState;
	ESQ						: ST_ITC_ESQ; // ITC message
	ECQ						: ST_ITC_ECQ; // ITC message
	MCQ						: ST_ITC_MCQ; // ITC message	
END_STRUCT
END_TYPE

// ---- 20_Product/10_BCF/11_Conv/13_Elements/01_DUTs/ST_ElementData.TcDUT
TYPE ST_ElementData :
(**************************************************************************************
 * 	Application		:	BoxControl Framework
 *	Revision		:	$Revision: 404529 $
 *	Revision date	:	$Date: 2018-04-23 08:21:38 +0200 (Mo., 23 Apr 2018) $
 *	Last changed by	:	$Author: b7bolm $
 *	URL				:	$URL: http://almscdc.swisslog.com/repo/SWPD/Development/BoxControlFramework/20_Release/trunk/01_Software/BCF/BCF/JumpStart/20_Product/10_App/13_Elements/10_Lib/10_Conv/01_DUTs/ST_ElementData.TcDUT $
 *
 *	Purpose			:	Element data - All data which are used internally. 
 *						External accessable over property (Read only)
 *
 * ------------------------------------------------------------------------------------
 *	Copyright Swisslog [IP AG], Switzerland. All rights reserved.
 * 
 * ------------------------------------------------------------------------------------
 *	
 * 	Revision History: 
 *
 * 	VERSION			DATE			INITIALS			DESCRIPTION
 *	0.1				01.01.2001		swl					Example
 *
 **************************************************************************************)
STRUCT
	Init					: BOOL; // Initialized
	InitRunning				: BOOL; // Init ongoing
	OperationState			: ST_PositionState; // Information about the state
	FunctionOrder			: ST_FunctionOrders; // Result of all functions
	MemberList				: ST_ElementMemberList; // List of objects which are linkt to this element
	ErrorData				: ST_ElementErrorStruct; // All error structures
	ControlRequest			: ST_ControlRequest; // Control request
END_STRUCT
END_TYPE

// ---- 20_Product/10_BCF/11_Conv/13_Elements/01_DUTs/ST_ElementErrorStruct.TcDUT
TYPE ST_ElementErrorStruct :
(**************************************************************************************
 * 	Application		:	BoxControl Framework
 *	Revision		:	$Revision: 404529 $
 *	Revision date	:	$Date: 2018-04-23 08:21:38 +0200 (Mo., 23 Apr 2018) $
 *	Last changed by	:	$Author: b7bolm $
 *	URL				:	$URL: http://almscdc.swisslog.com/repo/SWPD/Development/BoxControlFramework/20_Release/trunk/01_Software/BCF/BCF/JumpStart/20_Product/10_App/13_Elements/10_Lib/10_Conv/01_DUTs/ST_ElementErrorStruct.TcDUT $
 *
 *	Purpose			:	Element error structure - Contains all information for the
 *						error handling.
 *
 * ------------------------------------------------------------------------------------
 *	Copyright Swisslog [IP AG], Switzerland. All rights reserved.
 * 
 * ------------------------------------------------------------------------------------
 *	
 * 	Revision History: 
 *
 * 	VERSION			DATE			INITIALS			DESCRIPTION
 *	0.1				01.01.2001		swl					Example
 *
 **************************************************************************************)
STRUCT
	ErrorState				: E_ErrorState; // Ongoing module error state
	Error					: ST_ErrorDataSet; // Ongoing reported element error
	DataSetIdx				: INT; // Choosen error set index
	ErrorDataSet			: ARRAY [1..NUMBER_OF_ERROR_SETS] OF ST_ErrorDataSet; // Overview about all message sets
	ExternalError			: ST_ErrorDataSet; // External error, Can be set customized or by control code
	FunctionErrorPending	: BOOL; // An element function of this element is in error state
END_STRUCT
END_TYPE

// ---- 20_Product/10_BCF/11_Conv/13_Elements/01_DUTs/ST_ElementInterface.TcDUT
TYPE ST_ElementInterface :
(**************************************************************************************
 * 	Application		:	BoxControl Framework
 *	Revision		:	$Revision: 404529 $
 *	Revision date	:	$Date: 2018-04-23 08:21:38 +0200 (Mo., 23 Apr 2018) $
 *	Last changed by	:	$Author: b7bolm $
 *	URL				:	$URL: http://almscdc.swisslog.com/repo/SWPD/Development/BoxControlFramework/20_Release/trunk/01_Software/BCF/BCF/JumpStart/20_Product/10_App/13_Elements/10_Lib/10_Conv/01_DUTs/ST_ElementInterface.TcDUT $
 *
 *	Purpose			:	Element interface
 *
 * ------------------------------------------------------------------------------------
 *	Copyright Swisslog [IP AG], Switzerland. All rights reserved.
 * 
 * ------------------------------------------------------------------------------------
 *	
 * 	Revision History: 
 *
 * 	VERSION			DATE			INITIALS			DESCRIPTION
 *	0.1				01.01.2001		swl					Example
 *
 **************************************************************************************)
STRUCT
	In		: ST_ElementInterfaceIn;
	Out		: ST_ElementInterfaceOut;
END_STRUCT
END_TYPE

// ---- 20_Product/10_BCF/11_Conv/13_Elements/01_DUTs/ST_ElementInterfaceIn.TcDUT
TYPE ST_ElementInterfaceIn :
(**************************************************************************************
 * 	Application		:	BoxControl Framework
 *	Revision		:	$Revision: 404529 $
 *	Revision date	:	$Date: 2018-04-23 08:21:38 +0200 (Mo., 23 Apr 2018) $
 *	Last changed by	:	$Author: b7bolm $
 *	URL				:	$URL: http://almscdc.swisslog.com/repo/SWPD/Development/BoxControlFramework/20_Release/trunk/01_Software/BCF/BCF/JumpStart/20_Product/10_App/13_Elements/10_Lib/10_Conv/01_DUTs/ST_ElementInterfaceIn.TcDUT $
 *
 *	Purpose			:	Element data
 *
 * ------------------------------------------------------------------------------------
 *	Copyright Swisslog [IP AG], Switzerland. All rights reserved.
 * 
 * ------------------------------------------------------------------------------------
 *	
 * 	Revision History: 
 *
 * 	VERSION			DATE			INITIALS			DESCRIPTION
 *	0.1				01.01.2001		swl					Example
 *
 **************************************************************************************)	
STRUCT
	GroupState			: ST_PositionState;
	FunctionOrders		: ARRAY[1..Conveyor.NUMBER_OF_FUNCTIONS_PER_ELEMENT] OF ST_FunctionOrders;
	ElementStates		: ST_MasterSlaveStates;
	ElementEnable		: BOOL := TRUE; // External function enable 
END_STRUCT
END_TYPE

// ---- 20_Product/10_BCF/11_Conv/13_Elements/01_DUTs/ST_ElementInterfaceOut.TcDUT
TYPE ST_ElementInterfaceOut :
(**************************************************************************************
 * 	Application		:	BoxControl Framework
 *	Revision		:	$Revision: 404529 $
 *	Revision date	:	$Date: 2018-04-23 08:21:38 +0200 (Mo., 23 Apr 2018) $
 *	Last changed by	:	$Author: b7bolm $
 *	URL				:	$URL: http://almscdc.swisslog.com/repo/SWPD/Development/BoxControlFramework/20_Release/trunk/01_Software/BCF/BCF/JumpStart/20_Product/10_App/13_Elements/10_Lib/10_Conv/01_DUTs/ST_ElementInterfaceOut.TcDUT $
 *
 *	Purpose			:	Element data
 *
 * ------------------------------------------------------------------------------------
 *	Copyright Swisslog [IP AG], Switzerland. All rights reserved.
 * 
 * ------------------------------------------------------------------------------------
 *	
 * 	Revision History: 
 *
 * 	VERSION			DATE			INITIALS			DESCRIPTION
 *	0.1				01.01.2001		swl					Example
 *
 **************************************************************************************)	
STRUCT
	Interlock		: ST_Interlock; // Interlock structure
	State			: ST_ElementState; // Element states
END_STRUCT
END_TYPE

// ---- 20_Product/10_BCF/11_Conv/13_Elements/01_DUTs/ST_ElementMasterSlave.TcDUT
TYPE ST_ElementMasterSlave :
(**************************************************************************************
 * 	Application		:	BoxControl Framework
 *	Revision		:	$Revision: 404529 $
 *	Revision date	:	$Date: 2018-04-23 08:21:38 +0200 (Mo., 23 Apr 2018) $
 *	Last changed by	:	$Author: b7bolm $
 *	URL				:	$URL: http://almscdc.swisslog.com/repo/SWPD/Development/BoxControlFramework/20_Release/trunk/01_Software/BCF/BCF/JumpStart/20_Product/10_App/13_Elements/10_Lib/10_Conv/01_DUTs/ST_ElementMasterSlave.TcDUT $
 *
 *	Purpose			:	Master slave info
 *
 * ------------------------------------------------------------------------------------
 *	Copyright Swisslog [IP AG], Switzerland. All rights reserved.
 * 
 * ------------------------------------------------------------------------------------
 *	
 * 	Revision History: 
 *
 * 	VERSION			DATE			INITIALS			DESCRIPTION
 *	0.1				01.01.2001		swl					Example
 *
 **************************************************************************************)
STRUCT
	Master		: ST_ElementMasterSlaveEntry;
	Slave		: ST_ElementMasterSlaveEntry;
	Master_12	: ST_ElementMasterSlaveEntry;
	Slave_12	: ST_ElementMasterSlaveEntry;
	Master_34	: ST_ElementMasterSlaveEntry;
	Slave_34	: ST_ElementMasterSlaveEntry;

END_STRUCT
END_TYPE

// ---- 20_Product/10_BCF/11_Conv/13_Elements/01_DUTs/ST_ElementMasterSlaveEntry.TcDUT
TYPE ST_ElementMasterSlaveEntry :
(**************************************************************************************
 * 	Application		:	BoxControl Framework
 *	Revision		:	$Revision: 404529 $
 *	Revision date	:	$Date: 2018-04-23 08:21:38 +0200 (Mo., 23 Apr 2018) $
 *	Last changed by	:	$Author: b7bolm $
 *	URL				:	$URL: http://almscdc.swisslog.com/repo/SWPD/Development/BoxControlFramework/20_Release/trunk/01_Software/BCF/BCF/JumpStart/20_Product/10_App/13_Elements/10_Lib/10_Conv/01_DUTs/ST_ElementMasterSlaveEntry.TcDUT $
 *
 *	Purpose			:	Element slave
 *
 * ------------------------------------------------------------------------------------
 *	Copyright Swisslog [IP AG], Switzerland. All rights reserved.
 * 
 * ------------------------------------------------------------------------------------
 *	
 * 	Revision History: 
 *
 * 	VERSION			DATE			INITIALS			DESCRIPTION
 *	0.1				01.01.2001		swl					Example
 *
 **************************************************************************************)
STRUCT
	eElementNumber		: E_ElementNumber; // Linked element slave
END_STRUCT
END_TYPE

// ---- 20_Product/10_BCF/11_Conv/13_Elements/01_DUTs/ST_ElementMemberList.TcDUT
TYPE ST_ElementMemberList :
(**************************************************************************************
 * 	Application		:	BoxControl Framework
 *	Revision		:	$Revision: 404529 $
 *	Revision date	:	$Date: 2018-04-23 08:21:38 +0200 (Mo., 23 Apr 2018) $
 *	Last changed by	:	$Author: b7bolm $
 *	URL				:	$URL: http://almscdc.swisslog.com/repo/SWPD/Development/BoxControlFramework/20_Release/trunk/01_Software/BCF/BCF/JumpStart/20_Product/10_App/13_Elements/10_Lib/10_Conv/01_DUTs/ST_ElementMemberList.TcDUT $
 *
 *	Purpose			:	List of members which are linked to a element
 *
 * ------------------------------------------------------------------------------------
 *	Copyright Swisslog [IP AG], Switzerland. All rights reserved.
 * 
 * ------------------------------------------------------------------------------------
 *	
 * 	Revision History: 
 *
 * 	VERSION			DATE			INITIALS			DESCRIPTION
 *	0.1				01.01.2001		swl					Example
 *
 **************************************************************************************)
STRUCT
	FunctionList		: ARRAY [1 .. NUMBER_OF_FUNCTIONS_PER_ELEMENT] OF ST_FunctionEntry; // Registred function to this element
	ElementList			: ST_ElementMasterSlave; // Element slave
END_STRUCT
END_TYPE

// ---- 20_Product/10_BCF/11_Conv/13_Elements/01_DUTs/ST_ElementState.TcDUT
/// External element status - e.g. Master/Slave or function info, E.g. drive is running, element is in error state
TYPE ST_ElementState :
(**************************************************************************************
 *  Application     :   BoxControl Framework
 *  Revision date   :   $Date: 2013-09-23 11:26:06 +0200 (Wed, 23 Sep 2015) $
 *  Author          :   CDC
 * ------------------------------------------------------------------------------------
 *  © Swisslog AG
 *  Swisslog is not liable for any usage of this source code that is not agreed 
 *  on between Swisslog and the other party. The mandatory legal liability remains 
 *  unaffected.
 * ------------------------------------------------------------------------------------
 *  Revision History: 
 *
 *  VERSION DATE         INITIALS     DESCRIPTION
 *  0.0     DD.MM.YYYY   (name)       (explain customized modifications)
 *
 **************************************************************************************)
//Comment changed according to BCFD-6292 - ST_FunctionOrders, Comments not correct	
STRUCT
    //General
	Error			    : BOOL; // Element in error state
    
    //Axis 1 <-> 2
	DriveRunning	: BOOL; // Element drive is running
	DriveReady		: BOOL; // Drive is ready to start
    DriveDirection	: BOOL;	// Element drive direction TRUE = 1->2, False 2->1
	Speed			: INT; // Element uses this speed
	EncoderValue	: UINT; // Element encoder value
	
    //Axis 3 <-> 4
	DriveReady_34		: BOOL; // Drive is ready to start
	DriveRunning_34		: BOOL; // Element drive is running
    DriveDirection_34	: BOOL; // Element drive direction TRUE = 1->2, False 2->1
	Speed_34			: INT; // Element uses this speed		
    EncoderValue_34     : UINT; // Element encoder value
	
END_STRUCT
END_TYPE

// ---- 20_Product/10_BCF/11_Conv/13_Elements/01_DUTs/ST_FunctionEntry.TcDUT
TYPE ST_FunctionEntry :
(**************************************************************************************
 * 	Application		:	BoxControl Framework
 *	Revision		:	$Revision: 404529 $
 *	Revision date	:	$Date: 2018-04-23 08:21:38 +0200 (Mo., 23 Apr 2018) $
 *	Last changed by	:	$Author: b7bolm $
 *	URL				:	$URL: http://almscdc.swisslog.com/repo/SWPD/Development/BoxControlFramework/20_Release/trunk/01_Software/BCF/BCF/JumpStart/20_Product/10_App/13_Elements/10_Lib/10_Conv/01_DUTs/ST_FunctionEntry.TcDUT $
 *
 *	Purpose			:	Element functions
 *
 * ------------------------------------------------------------------------------------
 *	Copyright Swisslog [IP AG], Switzerland. All rights reserved.
 * 
 * ------------------------------------------------------------------------------------
 *	
 * 	Revision History: 
 *
 * 	VERSION			DATE			INITIALS			DESCRIPTION
 *	0.1				01.01.2001		swl					Example
 *
 **************************************************************************************)
STRUCT
	eFunctionNumber		: E_FunctionNumber; // Function number
END_STRUCT
END_TYPE

// ---- 20_Product/10_BCF/11_Conv/13_Elements/01_DUTs/ST_ITC_Element.TcDUT
TYPE ST_ITC_Element :
(**************************************************************************************
 * 	Application		:	BoxControl Framework
 *	Revision		:	$Revision: 404529 $
 *	Revision date	:	$Date: 2018-04-23 08:21:38 +0200 (Mo., 23 Apr 2018) $
 *	Last changed by	:	$Author: b7bolm $
 *	URL				:	$URL: http://almscdc.swisslog.com/repo/SWPD/Development/BoxControlFramework/20_Release/trunk/01_Software/BCF/BCF/JumpStart/20_Product/10_App/13_Elements/10_Lib/10_Conv/01_DUTs/ST_ITC_Element.TcDUT $
 *
 *	Purpose			:	Element ITC structure
 *
 * ------------------------------------------------------------------------------------
 *	Copyright Swisslog [IP AG], Switzerland. All rights reserved.
 * 
 * ------------------------------------------------------------------------------------
 *	
 * 	Revision History: 
 *
 * 	VERSION			DATE			INITIALS			DESCRIPTION
 *	0.1				01.01.2001		swl					Example
 *
 **************************************************************************************)
STRUCT
	Commands		: ST_ITC_ElementCommands; // Internal ITC commands
	Variable		: DINT; // Control variable
	ManualMotion	: ST_ITC_ManualMotion; // Command for manual motion
END_STRUCT
END_TYPE

// ---- 20_Product/10_BCF/11_Conv/13_Elements/01_DUTs/ST_ITC_ElementCommands.TcDUT
TYPE ST_ITC_ElementCommands :
(**************************************************************************************
 * 	Application		:	BoxControl Framework
 *	Revision		:	$Revision: 404529 $
 *	Revision date	:	$Date: 2018-04-23 08:21:38 +0200 (Mo., 23 Apr 2018) $
 *	Last changed by	:	$Author: b7bolm $
 *	URL				:	$URL: http://almscdc.swisslog.com/repo/SWPD/Development/BoxControlFramework/20_Release/trunk/01_Software/BCF/BCF/JumpStart/20_Product/10_App/13_Elements/10_Lib/10_Conv/01_DUTs/ST_ITC_ElementCommands.TcDUT $
 *
 *	Purpose			:	Internal ITC element commands
 *
 * ------------------------------------------------------------------------------------
 *	Copyright Swisslog [IP AG], Switzerland. All rights reserved.
 * 
 * ------------------------------------------------------------------------------------
 *	
 * 	Revision History: 
 *
 * 	VERSION			DATE			INITIALS			DESCRIPTION
 *	0.1				01.01.2001		swl					Example
 *
 **************************************************************************************)
STRUCT
	StatusReport		: BOOL; // Command to send StatusReport 
	ControlReport		: BOOL; // Command to send ControlReport 
	NoErrorReport		: BOOL; // Command to send a 'no error' report
	ManualControlReport	: BOOL; // Command to send a manual control report
END_STRUCT
END_TYPE

// ---- 20_Product/10_BCF/11_Conv/13_Elements/01_DUTs/ST_MasterSlaveStates.TcDUT
TYPE ST_MasterSlaveStates :
(**************************************************************************************
 * 	Application		:	BoxControl Framework
 *	Revision		:	$Revision: 404529 $
 *	Revision date	:	$Date: 2018-04-23 08:21:38 +0200 (Mo., 23 Apr 2018) $
 *	Last changed by	:	$Author: b7bolm $
 *	URL				:	$URL: http://almscdc.swisslog.com/repo/SWPD/Development/BoxControlFramework/20_Release/trunk/01_Software/BCF/BCF/JumpStart/20_Product/10_App/13_Elements/10_Lib/10_Conv/01_DUTs/ST_MasterSlaveStates.TcDUT $
 *
 *	Purpose			:	Master slave states
 *
 * ------------------------------------------------------------------------------------
 *	Copyright Swisslog [IP AG], Switzerland. All rights reserved.
 * 
 * ------------------------------------------------------------------------------------
 *	
 * 	Revision History: 
 *
 * 	VERSION			DATE			INITIALS			DESCRIPTION
 *	0.1				01.01.2001		swl					Example
 *
 **************************************************************************************)	
STRUCT
	Master 		: ST_ElementState;
	Slave		: ST_ElementState;
	Master_12	: ST_ElementState;
	Slave_12	: ST_ElementState;
	Master_34 	: ST_ElementState;
	Slave_34	: ST_ElementState;
END_STRUCT
END_TYPE

// ---- 20_Product/10_BCF/11_Conv/14_Groups/01_DUTs/E_GroupType.TcDUT
TYPE E_GroupType :
(**************************************************************************************
 * 	Application		:	BoxControl Framework
 *	Revision		:	$Revision: 404529 $
 *	Revision date	:	$Date: 2018-04-23 08:21:38 +0200 (Mo., 23 Apr 2018) $
 *	Last changed by	:	$Author: b7bolm $
 *	URL				:	$URL: http://almscdc.swisslog.com/repo/SWPD/Development/BoxControlFramework/20_Release/trunk/01_Software/BCF/BCF/JumpStart/20_Product/10_App/14_Groups/10_Lib/10_Conv/01_DUTs/E_GroupType.TcDUT $
 *
 *	Purpose			:	All available group types.
 *
 * ------------------------------------------------------------------------------------
 *	Copyright Swisslog [IP AG], Switzerland. All rights reserved.
 * 
 * ------------------------------------------------------------------------------------
 *	
 * 	Revision History: 
 *
 * 	VERSION			DATE			INITIALS			DESCRIPTION
 *	0.1				01.01.2001		swl					Example
 *
 **************************************************************************************)
(
	SG // Switching group
);
END_TYPE

// ---- 20_Product/10_BCF/11_Conv/14_Groups/01_DUTs/E_ITC_GroupControlCode.TcDUT
TYPE E_ITC_GroupControlCode :
(**************************************************************************************
 * 	Application		:	BoxControl Framework
 *	Revision		:	$Revision: 404529 $
 *	Revision date	:	$Date: 2018-04-23 08:21:38 +0200 (Mo., 23 Apr 2018) $
 *	Last changed by	:	$Author: b7bolm $
 *	URL				:	$URL: http://almscdc.swisslog.com/repo/SWPD/Development/BoxControlFramework/20_Release/trunk/01_Software/BCF/BCF/JumpStart/20_Product/10_App/14_Groups/10_Lib/10_Conv/01_DUTs/E_ITC_GroupControlCode.TcDUT $
 *
 *	Purpose			:	Group control code
 *
 * ------------------------------------------------------------------------------------
 *	Copyright Swisslog [IP AG], Switzerland. All rights reserved.
 * 
 * ------------------------------------------------------------------------------------
 *	
 * 	Revision History: 
 *
 * 	VERSION			DATE			INITIALS			DESCRIPTION
 *	0.1				01.01.2001		swl					Example
 *
 **************************************************************************************)
(
	NO_CODE					:= 0, // No code
	RESET_ERROR 			:= 1, // Acknowledge Error
	CHANGE_STATE 			:= 3, // E.g. start, stop
	CHANGE_MODE 			:= 4, // E.g. automatic, semiautomatic	
	SET_VARIABLE			:= 5  // Set Variable
);
END_TYPE

// ---- 20_Product/10_BCF/11_Conv/14_Groups/01_DUTs/ST_CFG_Group.TcDUT
TYPE ST_CFG_Group :
(**************************************************************************************
 * 	Application		:	BoxControl Framework
 *	Revision		:	$Revision: 404529 $
 *	Revision date	:	$Date: 2018-04-23 08:21:38 +0200 (Mo., 23 Apr 2018) $
 *	Last changed by	:	$Author: b7bolm $
 *	URL				:	$URL: http://almscdc.swisslog.com/repo/SWPD/Development/BoxControlFramework/20_Release/trunk/01_Software/BCF/BCF/JumpStart/20_Product/10_App/14_Groups/10_Lib/10_Conv/01_DUTs/10_Dummy/ST_CFG_Group.TcDUT $
 *
 *	Purpose			:	Config group
 *
 * ------------------------------------------------------------------------------------
 *	Copyright Swisslog [IP AG], Switzerland. All rights reserved.
 * 
 * ------------------------------------------------------------------------------------
 *	
 * 	Revision History: 
 *
 * 	VERSION			DATE			INITIALS			DESCRIPTION
 *	0.1				01.01.2001		swl					Example
 *
 **************************************************************************************)	
STRUCT
	GroupName				: STRING(NAME_LENGTH); // Group name
	eGroupNumber			: E_GroupNumber; // E-Number of the group
	eGroupType				: E_GroupType; // Group type
END_STRUCT
END_TYPE

// ---- 20_Product/10_BCF/11_Conv/14_Groups/01_DUTs/ST_GroupBase.TcDUT
TYPE ST_GroupBase :
(**************************************************************************************
 * 	Application		:	BoxControl Framework
 *	Revision		:	$Revision: 404529 $
 *	Revision date	:	$Date: 2018-04-23 08:21:38 +0200 (Mo., 23 Apr 2018) $
 *	Last changed by	:	$Author: b7bolm $
 *	URL				:	$URL: http://almscdc.swisslog.com/repo/SWPD/Development/BoxControlFramework/20_Release/trunk/01_Software/BCF/BCF/JumpStart/20_Product/10_App/14_Groups/10_Lib/10_Conv/01_DUTs/ST_GroupBase.TcDUT $
 *
 *	Purpose			:	Group base
 *
 * ------------------------------------------------------------------------------------
 *	Copyright Swisslog [IP AG], Switzerland. All rights reserved.
 * 
 * ------------------------------------------------------------------------------------
 *	
 * 	Revision History: 
 *
 * 	VERSION			DATE			INITIALS			DESCRIPTION
 *	0.1				01.01.2001		swl					Example
 *
 **************************************************************************************)
STRUCT
	eMsgType				: E_ITC_MsgTypeConv; // ITC msg type
	OperationStateEmpty		: ST_PositionState;
	GSQ						: ST_ITC_GSQ; // ITC Message
	GCQ						: ST_ITC_GCQ; // ITC Message
END_STRUCT
END_TYPE

// ---- 20_Product/10_BCF/11_Conv/14_Groups/01_DUTs/ST_GroupData.TcDUT
TYPE ST_GroupData :
(**************************************************************************************
 * 	Application		:	BoxControl Framework
 *	Revision		:	$Revision: 404529 $
 *	Revision date	:	$Date: 2018-04-23 08:21:38 +0200 (Mo., 23 Apr 2018) $
 *	Last changed by	:	$Author: b7bolm $
 *	URL				:	$URL: http://almscdc.swisslog.com/repo/SWPD/Development/BoxControlFramework/20_Release/trunk/01_Software/BCF/BCF/JumpStart/20_Product/10_App/14_Groups/10_Lib/10_Conv/01_DUTs/ST_GroupData.TcDUT $
 *
 *	Purpose			:	Group data - These datas are stored persistently.
 *
 * ------------------------------------------------------------------------------------
 *	Copyright Swisslog [IP AG], Switzerland. All rights reserved.
 * 
 * ------------------------------------------------------------------------------------
 *	
 * 	Revision History: 
 *
 * 	VERSION			DATE			INITIALS			DESCRIPTION
 *	0.1				01.01.2001		swl					Example
 *
 **************************************************************************************)
STRUCT
	Init				: BOOL; // Initialized
	InitRunning			: BOOL; // Init ongoing
	OperationState		: ST_PositionState; // Group state
	ErrorData			: ST_GroupErrorStruct; // Error data set 
END_STRUCT
END_TYPE

// ---- 20_Product/10_BCF/11_Conv/14_Groups/01_DUTs/ST_GroupErrorStruct.TcDUT
TYPE ST_GroupErrorStruct :
(**************************************************************************************
 * 	Application		:	BoxControl Framework
 *	Revision		:	$Revision: 404529 $
 *	Revision date	:	$Date: 2018-04-23 08:21:38 +0200 (Mo., 23 Apr 2018) $
 *	Last changed by	:	$Author: b7bolm $
 *	URL				:	$URL: http://almscdc.swisslog.com/repo/SWPD/Development/BoxControlFramework/20_Release/trunk/01_Software/BCF/BCF/JumpStart/20_Product/10_App/14_Groups/10_Lib/10_Conv/01_DUTs/ST_GroupErrorStruct.TcDUT $
 *
 *	Purpose			:	Group error structure - Contains all information for the
 *						error handling.
 *
 * ------------------------------------------------------------------------------------
 *	Copyright Swisslog [IP AG], Switzerland. All rights reserved.
 * 
 * ------------------------------------------------------------------------------------
 *	
 * 	Revision History: 
 *
 * 	VERSION			DATE			INITIALS			DESCRIPTION
 *	0.1				01.01.2001		swl					Example
 *
 **************************************************************************************)
STRUCT
	ErrorState				: E_ErrorState; // Ongoing module error state
	Error					: ST_ErrorDataSet; // Ongoing reported error
	DataSetIdx				: INT; // Choosen error set index
	ErrorDataSet			: ARRAY [1..NUMBER_OF_ERROR_SETS] OF ST_ErrorDataSet; // Overview about all message sets
	ExternalError			: ST_ErrorDataSet; // External error, Can be set customized or by control code
	ElementErrorPending		: BOOL; // An element of this group is in error state
END_STRUCT
END_TYPE

// ---- 20_Product/10_BCF/11_Conv/14_Groups/01_DUTs/ST_GroupInterface.TcDUT
TYPE ST_GroupInterface :
(**************************************************************************************
 * 	Application		:	BoxControl Framework
 *	Revision		:	$Revision: 404529 $
 *	Revision date	:	$Date: 2018-04-23 08:21:38 +0200 (Mo., 23 Apr 2018) $
 *	Last changed by	:	$Author: b7bolm $
 *	URL				:	$URL: http://almscdc.swisslog.com/repo/SWPD/Development/BoxControlFramework/20_Release/trunk/01_Software/BCF/BCF/JumpStart/20_Product/10_App/14_Groups/10_Lib/10_Conv/01_DUTs/ST_GroupInterface.TcDUT $
 *
 *	Purpose			:	Group interface - Data which has to be persistent and 
 *						read and writeable from outside.
 *
 * ------------------------------------------------------------------------------------
 *	Copyright Swisslog [IP AG], Switzerland. All rights reserved.
 * 
 * ------------------------------------------------------------------------------------
 *	
 * 	Revision History: 
 *
 * 	VERSION			DATE			INITIALS			DESCRIPTION
 *	0.1				01.01.2001		swl					Example
 *
 **************************************************************************************)
STRUCT
	In		: ST_GroupInterfaceIn;
	Out		: ST_GroupInterfaceOut;
END_STRUCT
END_TYPE

// ---- 20_Product/10_BCF/11_Conv/14_Groups/01_DUTs/ST_GroupInterfaceIn.TcDUT
TYPE ST_GroupInterfaceIn :
(**************************************************************************************
 * 	Application		:	BoxControl Framework
 *	Revision		:	$Revision: 404529 $
 *	Revision date	:	$Date: 2018-04-23 08:21:38 +0200 (Mo., 23 Apr 2018) $
 *	Last changed by	:	$Author: b7bolm $
 *	URL				:	$URL: http://almscdc.swisslog.com/repo/SWPD/Development/BoxControlFramework/20_Release/trunk/01_Software/BCF/BCF/JumpStart/20_Product/10_App/14_Groups/10_Lib/10_Conv/01_DUTs/ST_GroupInterfaceIn.TcDUT $
 *
 *	Purpose			:	Group interface - Data which has to be persistent and 
 *						read and writeable from outside.
 *
 * ------------------------------------------------------------------------------------
 *	Copyright Swisslog [IP AG], Switzerland. All rights reserved.
 * 
 * ------------------------------------------------------------------------------------
 *	
 * 	Revision History: 
 *
 * 	VERSION			DATE			INITIALS			DESCRIPTION
 *	0.1				01.01.2001		swl					Example
 *
 **************************************************************************************)
STRUCT
	SubsystemState			: ST_PositionState;
END_STRUCT
END_TYPE

// ---- 20_Product/10_BCF/11_Conv/14_Groups/01_DUTs/ST_GroupInterfaceOut.TcDUT
TYPE ST_GroupInterfaceOut :
(**************************************************************************************
 * 	Application		:	BoxControl Framework
 *	Revision		:	$Revision: 404529 $
 *	Revision date	:	$Date: 2018-04-23 08:21:38 +0200 (Mo., 23 Apr 2018) $
 *	Last changed by	:	$Author: b7bolm $
 *	URL				:	$URL: http://almscdc.swisslog.com/repo/SWPD/Development/BoxControlFramework/20_Release/trunk/01_Software/BCF/BCF/JumpStart/20_Product/10_App/14_Groups/10_Lib/10_Conv/01_DUTs/ST_GroupInterfaceOut.TcDUT $
 *
 *	Purpose			:	Group interface - Data which has to be persistent and 
 *						read and writeable from outside.
 *
 * ------------------------------------------------------------------------------------
 *	Copyright Swisslog [IP AG], Switzerland. All rights reserved.
 * 
 * ------------------------------------------------------------------------------------
 *	
 * 	Revision History: 
 *
 * 	VERSION			DATE			INITIALS			DESCRIPTION
 *	0.1				01.01.2001		swl					Example
 *
 **************************************************************************************)
STRUCT
	
END_STRUCT
END_TYPE

// ---- 20_Product/10_BCF/11_Conv/14_Groups/01_DUTs/ST_GroupManagerElementMember.TcDUT
TYPE ST_GroupManagerElementMember :
(**************************************************************************************
 * 	Application		:	BoxControl Framework
 *	Revision		:	$Revision: 404529 $
 *	Revision date	:	$Date: 2018-04-23 08:21:38 +0200 (Mo., 23 Apr 2018) $
 *	Last changed by	:	$Author: b7bolm $
 *	URL				:	$URL: http://almscdc.swisslog.com/repo/SWPD/Development/BoxControlFramework/20_Release/trunk/01_Software/BCF/BCF/JumpStart/20_Product/10_App/14_Groups/10_Lib/10_Conv/01_DUTs/ST_GroupManagerElementMember.TcDUT $
 *
 *	Purpose			:	Element member structure
 *
 * ------------------------------------------------------------------------------------
 *	Copyright Swisslog [IP AG], Switzerland. All rights reserved.
 * 
 * ------------------------------------------------------------------------------------
 *	
 * 	Revision History: 
 *
 * 	VERSION			DATE			INITIALS			DESCRIPTION
 *	0.1				01.01.2001		swl					Example
 *
 **************************************************************************************)
STRUCT
	eMemberElement	:ARRAY[E_BEGIN_ELEMENT..E_END_ELEMENT] OF E_ElementNumber; (* Associated elements *)
END_STRUCT
END_TYPE

// ---- 20_Product/10_BCF/11_Conv/14_Groups/01_DUTs/ST_GroupManagerGroupMember.TcDUT
TYPE ST_GroupManagerGroupMember :
(**************************************************************************************
 * 	Application		:	BoxControl Framework
 *	Revision		:	$Revision: 404529 $
 *	Revision date	:	$Date: 2018-04-23 08:21:38 +0200 (Mo., 23 Apr 2018) $
 *	Last changed by	:	$Author: b7bolm $
 *	URL				:	$URL: http://almscdc.swisslog.com/repo/SWPD/Development/BoxControlFramework/20_Release/trunk/01_Software/BCF/BCF/JumpStart/20_Product/10_App/14_Groups/10_Lib/10_Conv/01_DUTs/ST_GroupManagerGroupMember.TcDUT $
 *
 *	Purpose			:	Group member structure
 *
 * ------------------------------------------------------------------------------------
 *	Copyright Swisslog [IP AG], Switzerland. All rights reserved.
 * 
 * ------------------------------------------------------------------------------------
 *	
 * 	Revision History: 
 *
 * 	VERSION			DATE			INITIALS			DESCRIPTION
 *	0.1				01.01.2001		swl					Example
 *
 **************************************************************************************)
STRUCT
	eMemberGroup	:ARRAY[G_BEGIN_GROUP..G_END_GROUP] OF E_GroupNumber; (* Associated elements *)
END_STRUCT
END_TYPE

// ---- 20_Product/10_BCF/11_Conv/14_Groups/01_DUTs/ST_ITC_Group.TcDUT
TYPE ST_ITC_Group :
(**************************************************************************************
 * 	Application		:	BoxControl Framework
 *	Revision		:	$Revision: 404529 $
 *	Revision date	:	$Date: 2018-04-23 08:21:38 +0200 (Mo., 23 Apr 2018) $
 *	Last changed by	:	$Author: b7bolm $
 *	URL				:	$URL: http://almscdc.swisslog.com/repo/SWPD/Development/BoxControlFramework/20_Release/trunk/01_Software/BCF/BCF/JumpStart/20_Product/10_App/14_Groups/10_Lib/10_Conv/01_DUTs/ST_ITC_Group.TcDUT $
 *
 *	Purpose			:	Group ITC structure
 *
 * ------------------------------------------------------------------------------------
 *	Copyright Swisslog [IP AG], Switzerland. All rights reserved.
 * 
 * ------------------------------------------------------------------------------------
 *	
 * 	Revision History: 
 *
 * 	VERSION			DATE			INITIALS			DESCRIPTION
 *	0.1				01.01.2001		swl					Example
 *
 **************************************************************************************)
STRUCT
	Commands	: ST_ITC_GroupCommands; // Internal ITC commands
	Variable	: DINT; // Control variable
END_STRUCT
END_TYPE

// ---- 20_Product/10_BCF/11_Conv/14_Groups/01_DUTs/ST_ITC_GroupCommands.TcDUT
TYPE ST_ITC_GroupCommands :
(**************************************************************************************
 * 	Application		:	BoxControl Framework
 *	Revision		:	$Revision: 404529 $
 *	Revision date	:	$Date: 2018-04-23 08:21:38 +0200 (Mo., 23 Apr 2018) $
 *	Last changed by	:	$Author: b7bolm $
 *	URL				:	$URL: http://almscdc.swisslog.com/repo/SWPD/Development/BoxControlFramework/20_Release/trunk/01_Software/BCF/BCF/JumpStart/20_Product/10_App/14_Groups/10_Lib/10_Conv/01_DUTs/ST_ITC_GroupCommands.TcDUT $
 *
 *	Purpose			:	Internal ITC group commands
 *
 * ------------------------------------------------------------------------------------
 *	Copyright Swisslog [IP AG], Switzerland. All rights reserved.
 * 
 * ------------------------------------------------------------------------------------
 *	
 * 	Revision History: 
 *
 * 	VERSION			DATE			INITIALS			DESCRIPTION
 *	0.1				01.01.2001		swl					Example
 *
 **************************************************************************************)
STRUCT
	Start					: BOOL; // Command: Start group 
	Stop					: BOOL; // Command: Stop group
	eMode					: E_PositionMode; // Command: Requested mode
	NoErrorReport			: BOOL; // Command: Send no error report
	StatusReport			: BOOL; // Command: Send StatusReport
	ControlReport			: BOOL; // command: Send ControlReport
END_STRUCT
END_TYPE

// ---- 20_Product/10_BCF/11_Conv/14_Groups/01_DUTs/ST_ITC_GroupEmulation.TcDUT
TYPE ST_ITC_GroupEmulation :
(**************************************************************************************
 * 	Application		:	BoxControl Framework
 *	Revision		:	$Revision: 404529 $
 *	Revision date	:	$Date: 2018-04-23 08:21:38 +0200 (Mo., 23 Apr 2018) $
 *	Last changed by	:	$Author: b7bolm $
 *	URL				:	$URL: http://almscdc.swisslog.com/repo/SWPD/Development/BoxControlFramework/20_Release/trunk/01_Software/BCF/BCF/JumpStart/20_Product/11_Emu/14_Groups/10_Lib/10_Conv/01_DUTs/ST_ITC_GroupEmulation.TcDUT $
 *
 *	Purpose			:	Group ITC structures
 *
 * ------------------------------------------------------------------------------------
 *	Copyright Swisslog [IP AG], Switzerland. All rights reserved.
 * 
 * ------------------------------------------------------------------------------------
 *	
 * 	Revision History: 
 *
 * 	VERSION			DATE			INITIALS			DESCRIPTION
 *	0.1				01.01.2001		swl					Example
 *
 **************************************************************************************)
STRUCT
	Commands	: ST_ITC_GroupCommandsEmulation; // Internal group ITC commands
	
END_STRUCT
END_TYPE

// ---- 20_Product/10_BCF/11_Conv/15_Subsystem/01_DUTs/E_ITC_SubSystemControlCode.TcDUT
TYPE E_ITC_SubsystemControlCode :
(**************************************************************************************
 * 	Application		:	BoxControl Framework
 *	Revision		:	$Revision: 404529 $
 *	Revision date	:	$Date: 2018-04-23 08:21:38 +0200 (Mo., 23 Apr 2018) $
 *	Last changed by	:	$Author: b7bolm $
 *	URL				:	$URL: http://almscdc.swisslog.com/repo/SWPD/Development/BoxControlFramework/20_Release/trunk/01_Software/BCF/BCF/JumpStart/20_Product/10_App/15_Subsystem/10_Lib/10_Conv/01_DUTs/E_ITC_SubSystemControlCode.TcDUT $
 *
 *	Purpose			:	Subsystem control request code
 *
 * ------------------------------------------------------------------------------------
 *	Copyright Swisslog [IP AG], Switzerland. All rights reserved.
 * 
 * ------------------------------------------------------------------------------------
 *	
 * 	Revision History: 
 *
 * 	VERSION			DATE			INITIALS			DESCRIPTION
 *	0.1				01.01.2001		swl					Example
 *
 **************************************************************************************)
(
	NO_CODE							:= 0, // No code
	RESET_ERROR 					:= 1, // Reset Error
	SET_VARIABLE 					:= 5, // Set Variable
	SET_MASTER_SPEED				:= 6, // Set Subsystem master speed
	UPDATE_SYSTEM_TIME				:= 7, // Update system time
	REQUEST_GROUP_POSITION_STATUS	:= 8  // Request status of all groups and positions
);
END_TYPE

// ---- 20_Product/10_BCF/11_Conv/15_Subsystem/01_DUTs/E_SystemInfo.TcDUT
TYPE E_SystemInfo :
(**************************************************************************************
 * 	Application		:	BoxControl Framework
 *	Revision		:	$Revision: 404529 $
 *	Revision date	:	$Date: 2018-04-23 08:21:38 +0200 (Mo., 23 Apr 2018) $
 *	Last changed by	:	$Author: b7bolm $
 *	URL				:	$URL: http://almscdc.swisslog.com/repo/SWPD/Development/BoxControlFramework/20_Release/trunk/01_Software/BCF/BCF/JumpStart/20_Product/10_App/15_Subsystem/10_Lib/10_Conv/01_DUTs/E_SystemInfo.TcDUT $
 *
 *	Purpose			:	Subsystem system info
 *
 * ------------------------------------------------------------------------------------
 *	Copyright Swisslog [IP AG], Switzerland. All rights reserved.
 * 
 * ------------------------------------------------------------------------------------
 *	
 * 	Revision History: 
 *
 * 	VERSION			DATE			INITIALS			DESCRIPTION
 *	0.1				01.01.2001		swl					Example
 *
 **************************************************************************************)
(
	NO_INFO,
	RESTARTED,
	TIME_UPDATE_REQUIRED
);
END_TYPE

// ---- 20_Product/10_BCF/11_Conv/15_Subsystem/01_DUTs/ST_ITC_SubSystem.TcDUT
TYPE ST_ITC_Subsystem :
(**************************************************************************************
 * 	Application		:	BoxControl Framework
 *	Revision		:	$Revision: 404529 $
 *	Revision date	:	$Date: 2018-04-23 08:21:38 +0200 (Mo., 23 Apr 2018) $
 *	Last changed by	:	$Author: b7bolm $
 *	URL				:	$URL: http://almscdc.swisslog.com/repo/SWPD/Development/BoxControlFramework/20_Release/trunk/01_Software/BCF/BCF/JumpStart/20_Product/10_App/15_Subsystem/10_Lib/10_Conv/01_DUTs/ST_ITC_SubSystem.TcDUT $
 *
 *	Purpose			:	Subsystem ITC structure
 *
 * ------------------------------------------------------------------------------------
 *	Copyright Swisslog [IP AG], Switzerland. All rights reserved.
 * 
 * ------------------------------------------------------------------------------------
 *	
 * 	Revision History: 
 *
 * 	VERSION			DATE			INITIALS			DESCRIPTION
 *	0.1				01.01.2001		swl					Example
 *
 **************************************************************************************)
STRUCT
	Commands	: ST_ITC_SubsystemCommands; // Internal ITC commands
	Variable	: DINT; // Control variable
END_STRUCT
END_TYPE

// ---- 20_Product/10_BCF/11_Conv/15_Subsystem/01_DUTs/ST_ITC_SubSystemCommands.TcDUT
TYPE ST_ITC_SubsystemCommands :
(**************************************************************************************
 * 	Application		:	BoxControl Framework
 *	Revision		:	$Revision: 404529 $
 *	Revision date	:	$Date: 2018-04-23 08:21:38 +0200 (Mo., 23 Apr 2018) $
 *	Last changed by	:	$Author: b7bolm $
 *	URL				:	$URL: http://almscdc.swisslog.com/repo/SWPD/Development/BoxControlFramework/20_Release/trunk/01_Software/BCF/BCF/JumpStart/20_Product/10_App/15_Subsystem/10_Lib/10_Conv/01_DUTs/ST_ITC_SubSystemCommands.TcDUT $
 *
 *	Purpose			:	Subsystem ITC commands - Are set internally
 *
 * ------------------------------------------------------------------------------------
 *	Copyright Swisslog [IP AG], Switzerland. All rights reserved.
 * 
 * ------------------------------------------------------------------------------------
 *	
 * 	Revision History: 
 *
 * 	VERSION			DATE			INITIALS			DESCRIPTION
 *	0.1				01.01.2001		swl					Example
 *
 **************************************************************************************)
STRUCT
	SystemRestartInfo				: BOOL; // Command to send StatusReport after system restart
	RequestTimeUpdate				: BOOL; // Command to send StatusReport to request time update
	NoErrorReport					: BOOL; // Command to send StatusReport error is gone
	StatusReport					: BOOL; // Command to send default StatusReport
	ControlReport					: BOOL; // Command to send default ControlReport
	UpdateSystemTime				: BOOL; // Command to update system time internally
	UpdateAllGroupsAndPositions		: BOOL; // Command to send a full system status report
END_STRUCT
END_TYPE

// ---- 20_Product/10_BCF/11_Conv/15_Subsystem/01_DUTs/ST_SubSystemBase.TcDUT
TYPE ST_SubSystemBase :
(**************************************************************************************
 * 	Application		:	BoxControl Framework
 *	Revision		:	$Revision: 404529 $
 *	Revision date	:	$Date: 2018-04-23 08:21:38 +0200 (Mo., 23 Apr 2018) $
 *	Last changed by	:	$Author: b7bolm $
 *	URL				:	$URL: http://almscdc.swisslog.com/repo/SWPD/Development/BoxControlFramework/20_Release/trunk/01_Software/BCF/BCF/JumpStart/20_Product/10_App/15_Subsystem/10_Lib/10_Conv/01_DUTs/ST_SubSystemBase.TcDUT $
 *
 *	Purpose			:	Subsystem base data
 *
 * ------------------------------------------------------------------------------------
 *	Copyright Swisslog [IP AG], Switzerland. All rights reserved.
 * 
 * ------------------------------------------------------------------------------------
 *	
 * 	Revision History: 
 *
 * 	VERSION			DATE			INITIALS			DESCRIPTION
 *	0.1				01.01.2001		swl					Example
 *
 **************************************************************************************)
STRUCT
	SSQ							: ST_ITC_SSQ; // ITC Message
	SCQ							: ST_ITC_SCQ; // ITC Message
	GSQ							: ST_ITC_GSQ; // ITC Message
	ESQ							: ST_ITC_ESQ; // ITC Message
	FSQ							: ST_ITC_FSQ; // ITC Message
	TimeValue					: STRING; // Received time value
	eMsgType					: E_ITC_MsgTypeConv;
	eUpdateGroupNumber			: E_GroupNumber; // Groupnumber index for subsystem update
	eUpdateElementNumber		: E_ElementNumber; // Elementnumber index for subsystem update
	eUpdateFunctionNumber		: E_FunctionNumber; // FunctionNumber index for subsystem update
	UpdateGroupDone				: BOOL; // All status sent (Subsystem update) 
	UpdateElementDone			: BOOL; // All status sent (Subsystem update) 
	UpdateFunctionDone			: BOOL; // All status sent (Subsystem update) 
	UpdateChannelSrc			: E_MFCS_Channel; // Channel
	eLimitFunctionNumber		: E_FunctionNumber; // Initialization limit 
	eLimitElementNumber			: E_ElementNumber; // Initialization limit 
	eLimitGroupNumber			: E_GroupNumber; // Initialization limit 
	OperationStateEmpty			: ST_PositionState;
END_STRUCT
END_TYPE

